DATA_BLOCK "ACESYS_HMI_GROUP"   // DB2
TITLE = ACESYS GROUP DB
{ S7_Optimized_Access := 'FALSE' }
AUTHOR : METIS
FAMILY : ACESYS
NAME : GroupDB
VERSION : 8.0
   VAR
      STATUS : Array[0..500] of "ACESYS_HMI_STAT_32T";   // Group Status to HMI
   END_VAR
BEGIN
   STATUS[0].EXT.AlarmWarnUnAck := FALSE;
   STATUS[0].EXT.AckRequired := FALSE;
   STATUS[0].EXT.Maintanence := FALSE;
   STATUS[0].EXT.Operation := FALSE;
   STATUS[0].EXT.Forced := FALSE;
   STATUS[0].EXT.BIT29 := FALSE;
   STATUS[0].EXT.BIT30 := FALSE;
   STATUS[0].EXT.BIT31 := FALSE;
   STATUS[0].EXT.ModeBit1 := FALSE;
   STATUS[0].EXT.ModeBit2 := FALSE;
   STATUS[0].EXT.ModeBit3 := FALSE;
   STATUS[0].EXT.BIT19 := FALSE;
   STATUS[0].EXT.BIT20 := FALSE;
   STATUS[0].EXT.AlarmSuppressed := FALSE;
   STATUS[0].EXT.AlarmPresent := FALSE;
   STATUS[0].EXT.AlarmFailUnAck := FALSE;
   STATUS[0].Status := 0;
   STATUS[0].TimeStamp := 16#0000;
   STATUS[1].EXT.AlarmWarnUnAck := FALSE;
   STATUS[1].EXT.AckRequired := FALSE;
   STATUS[1].EXT.Maintanence := FALSE;
   STATUS[1].EXT.Operation := FALSE;
   STATUS[1].EXT.Forced := FALSE;
   STATUS[1].EXT.BIT29 := FALSE;
   STATUS[1].EXT.BIT30 := FALSE;
   STATUS[1].EXT.BIT31 := FALSE;
   STATUS[1].EXT.ModeBit1 := FALSE;
   STATUS[1].EXT.ModeBit2 := FALSE;
   STATUS[1].EXT.ModeBit3 := FALSE;
   STATUS[1].EXT.BIT19 := FALSE;
   STATUS[1].EXT.BIT20 := FALSE;
   STATUS[1].EXT.AlarmSuppressed := FALSE;
   STATUS[1].EXT.AlarmPresent := FALSE;
   STATUS[1].EXT.AlarmFailUnAck := FALSE;
   STATUS[1].Status := 8193;
   STATUS[1].TimeStamp := 16#CB75;
   STATUS[2].EXT.AlarmWarnUnAck := FALSE;
   STATUS[2].EXT.AckRequired := FALSE;
   STATUS[2].EXT.Maintanence := FALSE;
   STATUS[2].EXT.Operation := FALSE;
   STATUS[2].EXT.Forced := FALSE;
   STATUS[2].EXT.BIT29 := FALSE;
   STATUS[2].EXT.BIT30 := FALSE;
   STATUS[2].EXT.BIT31 := FALSE;
   STATUS[2].EXT.ModeBit1 := FALSE;
   STATUS[2].EXT.ModeBit2 := FALSE;
   STATUS[2].EXT.ModeBit3 := FALSE;
   STATUS[2].EXT.BIT19 := FALSE;
   STATUS[2].EXT.BIT20 := FALSE;
   STATUS[2].EXT.AlarmSuppressed := FALSE;
   STATUS[2].EXT.AlarmPresent := FALSE;
   STATUS[2].EXT.AlarmFailUnAck := FALSE;
   STATUS[2].Status := 8193;
   STATUS[2].TimeStamp := 16#E395;
   STATUS[3].EXT.AlarmWarnUnAck := FALSE;
   STATUS[3].EXT.AckRequired := FALSE;
   STATUS[3].EXT.Maintanence := FALSE;
   STATUS[3].EXT.Operation := FALSE;
   STATUS[3].EXT.Forced := FALSE;
   STATUS[3].EXT.BIT29 := FALSE;
   STATUS[3].EXT.BIT30 := FALSE;
   STATUS[3].EXT.BIT31 := FALSE;
   STATUS[3].EXT.ModeBit1 := FALSE;
   STATUS[3].EXT.ModeBit2 := FALSE;
   STATUS[3].EXT.ModeBit3 := FALSE;
   STATUS[3].EXT.BIT19 := FALSE;
   STATUS[3].EXT.BIT20 := FALSE;
   STATUS[3].EXT.AlarmSuppressed := FALSE;
   STATUS[3].EXT.AlarmPresent := FALSE;
   STATUS[3].EXT.AlarmFailUnAck := FALSE;
   STATUS[3].Status := 4286;
   STATUS[3].TimeStamp := 16#BB87;
   STATUS[4].EXT.AlarmWarnUnAck := FALSE;
   STATUS[4].EXT.AckRequired := FALSE;
   STATUS[4].EXT.Maintanence := FALSE;
   STATUS[4].EXT.Operation := FALSE;
   STATUS[4].EXT.Forced := FALSE;
   STATUS[4].EXT.BIT29 := FALSE;
   STATUS[4].EXT.BIT30 := FALSE;
   STATUS[4].EXT.BIT31 := FALSE;
   STATUS[4].EXT.ModeBit1 := FALSE;
   STATUS[4].EXT.ModeBit2 := FALSE;
   STATUS[4].EXT.ModeBit3 := FALSE;
   STATUS[4].EXT.BIT19 := FALSE;
   STATUS[4].EXT.BIT20 := FALSE;
   STATUS[4].EXT.AlarmSuppressed := FALSE;
   STATUS[4].EXT.AlarmPresent := FALSE;
   STATUS[4].EXT.AlarmFailUnAck := FALSE;
   STATUS[4].Status := 8215;
   STATUS[4].TimeStamp := 16#CB75;
   STATUS[5].EXT.AlarmWarnUnAck := FALSE;
   STATUS[5].EXT.AckRequired := FALSE;
   STATUS[5].EXT.Maintanence := FALSE;
   STATUS[5].EXT.Operation := FALSE;
   STATUS[5].EXT.Forced := FALSE;
   STATUS[5].EXT.BIT29 := FALSE;
   STATUS[5].EXT.BIT30 := FALSE;
   STATUS[5].EXT.BIT31 := FALSE;
   STATUS[5].EXT.ModeBit1 := FALSE;
   STATUS[5].EXT.ModeBit2 := FALSE;
   STATUS[5].EXT.ModeBit3 := FALSE;
   STATUS[5].EXT.BIT19 := FALSE;
   STATUS[5].EXT.BIT20 := FALSE;
   STATUS[5].EXT.AlarmSuppressed := FALSE;
   STATUS[5].EXT.AlarmPresent := FALSE;
   STATUS[5].EXT.AlarmFailUnAck := FALSE;
   STATUS[5].Status := 8193;
   STATUS[5].TimeStamp := 16#84C0;
   STATUS[6].EXT.AlarmWarnUnAck := FALSE;
   STATUS[6].EXT.AckRequired := FALSE;
   STATUS[6].EXT.Maintanence := FALSE;
   STATUS[6].EXT.Operation := FALSE;
   STATUS[6].EXT.Forced := FALSE;
   STATUS[6].EXT.BIT29 := FALSE;
   STATUS[6].EXT.BIT30 := FALSE;
   STATUS[6].EXT.BIT31 := FALSE;
   STATUS[6].EXT.ModeBit1 := FALSE;
   STATUS[6].EXT.ModeBit2 := FALSE;
   STATUS[6].EXT.ModeBit3 := FALSE;
   STATUS[6].EXT.BIT19 := FALSE;
   STATUS[6].EXT.BIT20 := FALSE;
   STATUS[6].EXT.AlarmSuppressed := FALSE;
   STATUS[6].EXT.AlarmPresent := FALSE;
   STATUS[6].EXT.AlarmFailUnAck := FALSE;
   STATUS[6].Status := 8193;
   STATUS[6].TimeStamp := 16#84BA;
   STATUS[7].EXT.AlarmWarnUnAck := FALSE;
   STATUS[7].EXT.AckRequired := FALSE;
   STATUS[7].EXT.Maintanence := FALSE;
   STATUS[7].EXT.Operation := TRUE;
   STATUS[7].EXT.Forced := FALSE;
   STATUS[7].EXT.BIT29 := FALSE;
   STATUS[7].EXT.BIT30 := FALSE;
   STATUS[7].EXT.BIT31 := FALSE;
   STATUS[7].EXT.ModeBit1 := FALSE;
   STATUS[7].EXT.ModeBit2 := FALSE;
   STATUS[7].EXT.ModeBit3 := FALSE;
   STATUS[7].EXT.BIT19 := FALSE;
   STATUS[7].EXT.BIT20 := FALSE;
   STATUS[7].EXT.AlarmSuppressed := FALSE;
   STATUS[7].EXT.AlarmPresent := FALSE;
   STATUS[7].EXT.AlarmFailUnAck := FALSE;
   STATUS[7].Status := 4104;
   STATUS[7].TimeStamp := 16#C030;
   STATUS[8].EXT.AlarmWarnUnAck := FALSE;
   STATUS[8].EXT.AckRequired := FALSE;
   STATUS[8].EXT.Maintanence := FALSE;
   STATUS[8].EXT.Operation := FALSE;
   STATUS[8].EXT.Forced := FALSE;
   STATUS[8].EXT.BIT29 := FALSE;
   STATUS[8].EXT.BIT30 := FALSE;
   STATUS[8].EXT.BIT31 := FALSE;
   STATUS[8].EXT.ModeBit1 := FALSE;
   STATUS[8].EXT.ModeBit2 := FALSE;
   STATUS[8].EXT.ModeBit3 := FALSE;
   STATUS[8].EXT.BIT19 := FALSE;
   STATUS[8].EXT.BIT20 := FALSE;
   STATUS[8].EXT.AlarmSuppressed := FALSE;
   STATUS[8].EXT.AlarmPresent := FALSE;
   STATUS[8].EXT.AlarmFailUnAck := FALSE;
   STATUS[8].Status := 8193;
   STATUS[8].TimeStamp := 16#60BB;
   STATUS[9].EXT.AlarmWarnUnAck := FALSE;
   STATUS[9].EXT.AckRequired := FALSE;
   STATUS[9].EXT.Maintanence := FALSE;
   STATUS[9].EXT.Operation := FALSE;
   STATUS[9].EXT.Forced := FALSE;
   STATUS[9].EXT.BIT29 := FALSE;
   STATUS[9].EXT.BIT30 := FALSE;
   STATUS[9].EXT.BIT31 := FALSE;
   STATUS[9].EXT.ModeBit1 := FALSE;
   STATUS[9].EXT.ModeBit2 := FALSE;
   STATUS[9].EXT.ModeBit3 := FALSE;
   STATUS[9].EXT.BIT19 := FALSE;
   STATUS[9].EXT.BIT20 := FALSE;
   STATUS[9].EXT.AlarmSuppressed := FALSE;
   STATUS[9].EXT.AlarmPresent := FALSE;
   STATUS[9].EXT.AlarmFailUnAck := FALSE;
   STATUS[9].Status := 8193;
   STATUS[9].TimeStamp := 16#60BB;
   STATUS[10].EXT.AlarmWarnUnAck := FALSE;
   STATUS[10].EXT.AckRequired := FALSE;
   STATUS[10].EXT.Maintanence := FALSE;
   STATUS[10].EXT.Operation := FALSE;
   STATUS[10].EXT.Forced := FALSE;
   STATUS[10].EXT.BIT29 := FALSE;
   STATUS[10].EXT.BIT30 := FALSE;
   STATUS[10].EXT.BIT31 := FALSE;
   STATUS[10].EXT.ModeBit1 := FALSE;
   STATUS[10].EXT.ModeBit2 := FALSE;
   STATUS[10].EXT.ModeBit3 := FALSE;
   STATUS[10].EXT.BIT19 := FALSE;
   STATUS[10].EXT.BIT20 := FALSE;
   STATUS[10].EXT.AlarmSuppressed := FALSE;
   STATUS[10].EXT.AlarmPresent := FALSE;
   STATUS[10].EXT.AlarmFailUnAck := FALSE;
   STATUS[10].Status := 8193;
   STATUS[10].TimeStamp := 16#60BB;
   STATUS[11].EXT.AlarmWarnUnAck := FALSE;
   STATUS[11].EXT.AckRequired := FALSE;
   STATUS[11].EXT.Maintanence := FALSE;
   STATUS[11].EXT.Operation := FALSE;
   STATUS[11].EXT.Forced := FALSE;
   STATUS[11].EXT.BIT29 := FALSE;
   STATUS[11].EXT.BIT30 := FALSE;
   STATUS[11].EXT.BIT31 := FALSE;
   STATUS[11].EXT.ModeBit1 := FALSE;
   STATUS[11].EXT.ModeBit2 := FALSE;
   STATUS[11].EXT.ModeBit3 := FALSE;
   STATUS[11].EXT.BIT19 := FALSE;
   STATUS[11].EXT.BIT20 := FALSE;
   STATUS[11].EXT.AlarmSuppressed := FALSE;
   STATUS[11].EXT.AlarmPresent := FALSE;
   STATUS[11].EXT.AlarmFailUnAck := FALSE;
   STATUS[11].Status := 8193;
   STATUS[11].TimeStamp := 16#60BB;
   STATUS[12].EXT.AlarmWarnUnAck := FALSE;
   STATUS[12].EXT.AckRequired := FALSE;
   STATUS[12].EXT.Maintanence := FALSE;
   STATUS[12].EXT.Operation := FALSE;
   STATUS[12].EXT.Forced := FALSE;
   STATUS[12].EXT.BIT29 := FALSE;
   STATUS[12].EXT.BIT30 := FALSE;
   STATUS[12].EXT.BIT31 := FALSE;
   STATUS[12].EXT.ModeBit1 := FALSE;
   STATUS[12].EXT.ModeBit2 := FALSE;
   STATUS[12].EXT.ModeBit3 := FALSE;
   STATUS[12].EXT.BIT19 := FALSE;
   STATUS[12].EXT.BIT20 := FALSE;
   STATUS[12].EXT.AlarmSuppressed := FALSE;
   STATUS[12].EXT.AlarmPresent := FALSE;
   STATUS[12].EXT.AlarmFailUnAck := FALSE;
   STATUS[12].Status := 8193;
   STATUS[12].TimeStamp := 16#60BB;
   STATUS[13].EXT.AlarmWarnUnAck := FALSE;
   STATUS[13].EXT.AckRequired := FALSE;
   STATUS[13].EXT.Maintanence := FALSE;
   STATUS[13].EXT.Operation := FALSE;
   STATUS[13].EXT.Forced := FALSE;
   STATUS[13].EXT.BIT29 := FALSE;
   STATUS[13].EXT.BIT30 := FALSE;
   STATUS[13].EXT.BIT31 := FALSE;
   STATUS[13].EXT.ModeBit1 := FALSE;
   STATUS[13].EXT.ModeBit2 := FALSE;
   STATUS[13].EXT.ModeBit3 := FALSE;
   STATUS[13].EXT.BIT19 := FALSE;
   STATUS[13].EXT.BIT20 := FALSE;
   STATUS[13].EXT.AlarmSuppressed := FALSE;
   STATUS[13].EXT.AlarmPresent := FALSE;
   STATUS[13].EXT.AlarmFailUnAck := FALSE;
   STATUS[13].Status := 8193;
   STATUS[13].TimeStamp := 16#60BB;
   STATUS[14].EXT.AlarmWarnUnAck := FALSE;
   STATUS[14].EXT.AckRequired := FALSE;
   STATUS[14].EXT.Maintanence := FALSE;
   STATUS[14].EXT.Operation := FALSE;
   STATUS[14].EXT.Forced := FALSE;
   STATUS[14].EXT.BIT29 := FALSE;
   STATUS[14].EXT.BIT30 := FALSE;
   STATUS[14].EXT.BIT31 := FALSE;
   STATUS[14].EXT.ModeBit1 := FALSE;
   STATUS[14].EXT.ModeBit2 := FALSE;
   STATUS[14].EXT.ModeBit3 := FALSE;
   STATUS[14].EXT.BIT19 := FALSE;
   STATUS[14].EXT.BIT20 := FALSE;
   STATUS[14].EXT.AlarmSuppressed := FALSE;
   STATUS[14].EXT.AlarmPresent := FALSE;
   STATUS[14].EXT.AlarmFailUnAck := FALSE;
   STATUS[14].Status := 8193;
   STATUS[14].TimeStamp := 16#60BB;
   STATUS[15].EXT.AlarmWarnUnAck := FALSE;
   STATUS[15].EXT.AckRequired := FALSE;
   STATUS[15].EXT.Maintanence := FALSE;
   STATUS[15].EXT.Operation := FALSE;
   STATUS[15].EXT.Forced := FALSE;
   STATUS[15].EXT.BIT29 := FALSE;
   STATUS[15].EXT.BIT30 := FALSE;
   STATUS[15].EXT.BIT31 := FALSE;
   STATUS[15].EXT.ModeBit1 := FALSE;
   STATUS[15].EXT.ModeBit2 := FALSE;
   STATUS[15].EXT.ModeBit3 := FALSE;
   STATUS[15].EXT.BIT19 := FALSE;
   STATUS[15].EXT.BIT20 := FALSE;
   STATUS[15].EXT.AlarmSuppressed := FALSE;
   STATUS[15].EXT.AlarmPresent := FALSE;
   STATUS[15].EXT.AlarmFailUnAck := FALSE;
   STATUS[15].Status := 8193;
   STATUS[15].TimeStamp := 16#60BB;
   STATUS[16].EXT.AlarmWarnUnAck := FALSE;
   STATUS[16].EXT.AckRequired := FALSE;
   STATUS[16].EXT.Maintanence := FALSE;
   STATUS[16].EXT.Operation := FALSE;
   STATUS[16].EXT.Forced := FALSE;
   STATUS[16].EXT.BIT29 := FALSE;
   STATUS[16].EXT.BIT30 := FALSE;
   STATUS[16].EXT.BIT31 := FALSE;
   STATUS[16].EXT.ModeBit1 := FALSE;
   STATUS[16].EXT.ModeBit2 := FALSE;
   STATUS[16].EXT.ModeBit3 := FALSE;
   STATUS[16].EXT.BIT19 := FALSE;
   STATUS[16].EXT.BIT20 := FALSE;
   STATUS[16].EXT.AlarmSuppressed := FALSE;
   STATUS[16].EXT.AlarmPresent := FALSE;
   STATUS[16].EXT.AlarmFailUnAck := FALSE;
   STATUS[16].Status := 0;
   STATUS[16].TimeStamp := 16#0000;
   STATUS[17].EXT.AlarmWarnUnAck := FALSE;
   STATUS[17].EXT.AckRequired := FALSE;
   STATUS[17].EXT.Maintanence := FALSE;
   STATUS[17].EXT.Operation := FALSE;
   STATUS[17].EXT.Forced := FALSE;
   STATUS[17].EXT.BIT29 := FALSE;
   STATUS[17].EXT.BIT30 := FALSE;
   STATUS[17].EXT.BIT31 := FALSE;
   STATUS[17].EXT.ModeBit1 := FALSE;
   STATUS[17].EXT.ModeBit2 := FALSE;
   STATUS[17].EXT.ModeBit3 := FALSE;
   STATUS[17].EXT.BIT19 := FALSE;
   STATUS[17].EXT.BIT20 := FALSE;
   STATUS[17].EXT.AlarmSuppressed := FALSE;
   STATUS[17].EXT.AlarmPresent := FALSE;
   STATUS[17].EXT.AlarmFailUnAck := FALSE;
   STATUS[17].Status := 0;
   STATUS[17].TimeStamp := 16#0000;
   STATUS[18].EXT.AlarmWarnUnAck := FALSE;
   STATUS[18].EXT.AckRequired := FALSE;
   STATUS[18].EXT.Maintanence := FALSE;
   STATUS[18].EXT.Operation := FALSE;
   STATUS[18].EXT.Forced := FALSE;
   STATUS[18].EXT.BIT29 := FALSE;
   STATUS[18].EXT.BIT30 := FALSE;
   STATUS[18].EXT.BIT31 := FALSE;
   STATUS[18].EXT.ModeBit1 := FALSE;
   STATUS[18].EXT.ModeBit2 := FALSE;
   STATUS[18].EXT.ModeBit3 := FALSE;
   STATUS[18].EXT.BIT19 := FALSE;
   STATUS[18].EXT.BIT20 := FALSE;
   STATUS[18].EXT.AlarmSuppressed := FALSE;
   STATUS[18].EXT.AlarmPresent := FALSE;
   STATUS[18].EXT.AlarmFailUnAck := FALSE;
   STATUS[18].Status := 0;
   STATUS[18].TimeStamp := 16#0000;
   STATUS[19].EXT.AlarmWarnUnAck := FALSE;
   STATUS[19].EXT.AckRequired := FALSE;
   STATUS[19].EXT.Maintanence := FALSE;
   STATUS[19].EXT.Operation := FALSE;
   STATUS[19].EXT.Forced := FALSE;
   STATUS[19].EXT.BIT29 := FALSE;
   STATUS[19].EXT.BIT30 := FALSE;
   STATUS[19].EXT.BIT31 := FALSE;
   STATUS[19].EXT.ModeBit1 := FALSE;
   STATUS[19].EXT.ModeBit2 := FALSE;
   STATUS[19].EXT.ModeBit3 := FALSE;
   STATUS[19].EXT.BIT19 := FALSE;
   STATUS[19].EXT.BIT20 := FALSE;
   STATUS[19].EXT.AlarmSuppressed := FALSE;
   STATUS[19].EXT.AlarmPresent := FALSE;
   STATUS[19].EXT.AlarmFailUnAck := FALSE;
   STATUS[19].Status := 0;
   STATUS[19].TimeStamp := 16#0000;
   STATUS[20].EXT.AlarmWarnUnAck := FALSE;
   STATUS[20].EXT.AckRequired := FALSE;
   STATUS[20].EXT.Maintanence := FALSE;
   STATUS[20].EXT.Operation := FALSE;
   STATUS[20].EXT.Forced := FALSE;
   STATUS[20].EXT.BIT29 := FALSE;
   STATUS[20].EXT.BIT30 := FALSE;
   STATUS[20].EXT.BIT31 := FALSE;
   STATUS[20].EXT.ModeBit1 := FALSE;
   STATUS[20].EXT.ModeBit2 := FALSE;
   STATUS[20].EXT.ModeBit3 := FALSE;
   STATUS[20].EXT.BIT19 := FALSE;
   STATUS[20].EXT.BIT20 := FALSE;
   STATUS[20].EXT.AlarmSuppressed := FALSE;
   STATUS[20].EXT.AlarmPresent := FALSE;
   STATUS[20].EXT.AlarmFailUnAck := FALSE;
   STATUS[20].Status := 0;
   STATUS[20].TimeStamp := 16#0000;
   STATUS[21].EXT.AlarmWarnUnAck := FALSE;
   STATUS[21].EXT.AckRequired := FALSE;
   STATUS[21].EXT.Maintanence := FALSE;
   STATUS[21].EXT.Operation := FALSE;
   STATUS[21].EXT.Forced := FALSE;
   STATUS[21].EXT.BIT29 := FALSE;
   STATUS[21].EXT.BIT30 := FALSE;
   STATUS[21].EXT.BIT31 := FALSE;
   STATUS[21].EXT.ModeBit1 := FALSE;
   STATUS[21].EXT.ModeBit2 := FALSE;
   STATUS[21].EXT.ModeBit3 := FALSE;
   STATUS[21].EXT.BIT19 := FALSE;
   STATUS[21].EXT.BIT20 := FALSE;
   STATUS[21].EXT.AlarmSuppressed := FALSE;
   STATUS[21].EXT.AlarmPresent := FALSE;
   STATUS[21].EXT.AlarmFailUnAck := FALSE;
   STATUS[21].Status := 0;
   STATUS[21].TimeStamp := 16#0000;
   STATUS[22].EXT.AlarmWarnUnAck := FALSE;
   STATUS[22].EXT.AckRequired := FALSE;
   STATUS[22].EXT.Maintanence := FALSE;
   STATUS[22].EXT.Operation := FALSE;
   STATUS[22].EXT.Forced := FALSE;
   STATUS[22].EXT.BIT29 := FALSE;
   STATUS[22].EXT.BIT30 := FALSE;
   STATUS[22].EXT.BIT31 := FALSE;
   STATUS[22].EXT.ModeBit1 := FALSE;
   STATUS[22].EXT.ModeBit2 := FALSE;
   STATUS[22].EXT.ModeBit3 := FALSE;
   STATUS[22].EXT.BIT19 := FALSE;
   STATUS[22].EXT.BIT20 := FALSE;
   STATUS[22].EXT.AlarmSuppressed := FALSE;
   STATUS[22].EXT.AlarmPresent := FALSE;
   STATUS[22].EXT.AlarmFailUnAck := FALSE;
   STATUS[22].Status := 0;
   STATUS[22].TimeStamp := 16#0000;
   STATUS[23].EXT.AlarmWarnUnAck := FALSE;
   STATUS[23].EXT.AckRequired := FALSE;
   STATUS[23].EXT.Maintanence := FALSE;
   STATUS[23].EXT.Operation := FALSE;
   STATUS[23].EXT.Forced := FALSE;
   STATUS[23].EXT.BIT29 := FALSE;
   STATUS[23].EXT.BIT30 := FALSE;
   STATUS[23].EXT.BIT31 := FALSE;
   STATUS[23].EXT.ModeBit1 := FALSE;
   STATUS[23].EXT.ModeBit2 := FALSE;
   STATUS[23].EXT.ModeBit3 := FALSE;
   STATUS[23].EXT.BIT19 := FALSE;
   STATUS[23].EXT.BIT20 := FALSE;
   STATUS[23].EXT.AlarmSuppressed := FALSE;
   STATUS[23].EXT.AlarmPresent := FALSE;
   STATUS[23].EXT.AlarmFailUnAck := FALSE;
   STATUS[23].Status := 0;
   STATUS[23].TimeStamp := 16#0000;
   STATUS[24].EXT.AlarmWarnUnAck := FALSE;
   STATUS[24].EXT.AckRequired := FALSE;
   STATUS[24].EXT.Maintanence := FALSE;
   STATUS[24].EXT.Operation := FALSE;
   STATUS[24].EXT.Forced := FALSE;
   STATUS[24].EXT.BIT29 := FALSE;
   STATUS[24].EXT.BIT30 := FALSE;
   STATUS[24].EXT.BIT31 := FALSE;
   STATUS[24].EXT.ModeBit1 := FALSE;
   STATUS[24].EXT.ModeBit2 := FALSE;
   STATUS[24].EXT.ModeBit3 := FALSE;
   STATUS[24].EXT.BIT19 := FALSE;
   STATUS[24].EXT.BIT20 := FALSE;
   STATUS[24].EXT.AlarmSuppressed := FALSE;
   STATUS[24].EXT.AlarmPresent := FALSE;
   STATUS[24].EXT.AlarmFailUnAck := FALSE;
   STATUS[24].Status := 0;
   STATUS[24].TimeStamp := 16#0000;
   STATUS[25].EXT.AlarmWarnUnAck := FALSE;
   STATUS[25].EXT.AckRequired := FALSE;
   STATUS[25].EXT.Maintanence := FALSE;
   STATUS[25].EXT.Operation := FALSE;
   STATUS[25].EXT.Forced := FALSE;
   STATUS[25].EXT.BIT29 := FALSE;
   STATUS[25].EXT.BIT30 := FALSE;
   STATUS[25].EXT.BIT31 := FALSE;
   STATUS[25].EXT.ModeBit1 := FALSE;
   STATUS[25].EXT.ModeBit2 := FALSE;
   STATUS[25].EXT.ModeBit3 := FALSE;
   STATUS[25].EXT.BIT19 := FALSE;
   STATUS[25].EXT.BIT20 := FALSE;
   STATUS[25].EXT.AlarmSuppressed := FALSE;
   STATUS[25].EXT.AlarmPresent := FALSE;
   STATUS[25].EXT.AlarmFailUnAck := FALSE;
   STATUS[25].Status := 0;
   STATUS[25].TimeStamp := 16#0000;
   STATUS[26].EXT.AlarmWarnUnAck := FALSE;
   STATUS[26].EXT.AckRequired := FALSE;
   STATUS[26].EXT.Maintanence := FALSE;
   STATUS[26].EXT.Operation := FALSE;
   STATUS[26].EXT.Forced := FALSE;
   STATUS[26].EXT.BIT29 := FALSE;
   STATUS[26].EXT.BIT30 := FALSE;
   STATUS[26].EXT.BIT31 := FALSE;
   STATUS[26].EXT.ModeBit1 := FALSE;
   STATUS[26].EXT.ModeBit2 := FALSE;
   STATUS[26].EXT.ModeBit3 := FALSE;
   STATUS[26].EXT.BIT19 := FALSE;
   STATUS[26].EXT.BIT20 := FALSE;
   STATUS[26].EXT.AlarmSuppressed := FALSE;
   STATUS[26].EXT.AlarmPresent := FALSE;
   STATUS[26].EXT.AlarmFailUnAck := FALSE;
   STATUS[26].Status := 0;
   STATUS[26].TimeStamp := 16#0000;
   STATUS[27].EXT.AlarmWarnUnAck := FALSE;
   STATUS[27].EXT.AckRequired := FALSE;
   STATUS[27].EXT.Maintanence := FALSE;
   STATUS[27].EXT.Operation := FALSE;
   STATUS[27].EXT.Forced := FALSE;
   STATUS[27].EXT.BIT29 := FALSE;
   STATUS[27].EXT.BIT30 := FALSE;
   STATUS[27].EXT.BIT31 := FALSE;
   STATUS[27].EXT.ModeBit1 := FALSE;
   STATUS[27].EXT.ModeBit2 := FALSE;
   STATUS[27].EXT.ModeBit3 := FALSE;
   STATUS[27].EXT.BIT19 := FALSE;
   STATUS[27].EXT.BIT20 := FALSE;
   STATUS[27].EXT.AlarmSuppressed := FALSE;
   STATUS[27].EXT.AlarmPresent := FALSE;
   STATUS[27].EXT.AlarmFailUnAck := FALSE;
   STATUS[27].Status := 0;
   STATUS[27].TimeStamp := 16#0000;
   STATUS[28].EXT.AlarmWarnUnAck := FALSE;
   STATUS[28].EXT.AckRequired := FALSE;
   STATUS[28].EXT.Maintanence := FALSE;
   STATUS[28].EXT.Operation := FALSE;
   STATUS[28].EXT.Forced := FALSE;
   STATUS[28].EXT.BIT29 := FALSE;
   STATUS[28].EXT.BIT30 := FALSE;
   STATUS[28].EXT.BIT31 := FALSE;
   STATUS[28].EXT.ModeBit1 := FALSE;
   STATUS[28].EXT.ModeBit2 := FALSE;
   STATUS[28].EXT.ModeBit3 := FALSE;
   STATUS[28].EXT.BIT19 := FALSE;
   STATUS[28].EXT.BIT20 := FALSE;
   STATUS[28].EXT.AlarmSuppressed := FALSE;
   STATUS[28].EXT.AlarmPresent := FALSE;
   STATUS[28].EXT.AlarmFailUnAck := FALSE;
   STATUS[28].Status := 0;
   STATUS[28].TimeStamp := 16#0000;
   STATUS[29].EXT.AlarmWarnUnAck := FALSE;
   STATUS[29].EXT.AckRequired := FALSE;
   STATUS[29].EXT.Maintanence := FALSE;
   STATUS[29].EXT.Operation := FALSE;
   STATUS[29].EXT.Forced := FALSE;
   STATUS[29].EXT.BIT29 := FALSE;
   STATUS[29].EXT.BIT30 := FALSE;
   STATUS[29].EXT.BIT31 := FALSE;
   STATUS[29].EXT.ModeBit1 := FALSE;
   STATUS[29].EXT.ModeBit2 := FALSE;
   STATUS[29].EXT.ModeBit3 := FALSE;
   STATUS[29].EXT.BIT19 := FALSE;
   STATUS[29].EXT.BIT20 := FALSE;
   STATUS[29].EXT.AlarmSuppressed := FALSE;
   STATUS[29].EXT.AlarmPresent := FALSE;
   STATUS[29].EXT.AlarmFailUnAck := FALSE;
   STATUS[29].Status := 0;
   STATUS[29].TimeStamp := 16#0000;
   STATUS[30].EXT.AlarmWarnUnAck := FALSE;
   STATUS[30].EXT.AckRequired := FALSE;
   STATUS[30].EXT.Maintanence := FALSE;
   STATUS[30].EXT.Operation := FALSE;
   STATUS[30].EXT.Forced := FALSE;
   STATUS[30].EXT.BIT29 := FALSE;
   STATUS[30].EXT.BIT30 := FALSE;
   STATUS[30].EXT.BIT31 := FALSE;
   STATUS[30].EXT.ModeBit1 := FALSE;
   STATUS[30].EXT.ModeBit2 := FALSE;
   STATUS[30].EXT.ModeBit3 := FALSE;
   STATUS[30].EXT.BIT19 := FALSE;
   STATUS[30].EXT.BIT20 := FALSE;
   STATUS[30].EXT.AlarmSuppressed := FALSE;
   STATUS[30].EXT.AlarmPresent := FALSE;
   STATUS[30].EXT.AlarmFailUnAck := FALSE;
   STATUS[30].Status := 0;
   STATUS[30].TimeStamp := 16#0000;
   STATUS[31].EXT.AlarmWarnUnAck := FALSE;
   STATUS[31].EXT.AckRequired := FALSE;
   STATUS[31].EXT.Maintanence := FALSE;
   STATUS[31].EXT.Operation := FALSE;
   STATUS[31].EXT.Forced := FALSE;
   STATUS[31].EXT.BIT29 := FALSE;
   STATUS[31].EXT.BIT30 := FALSE;
   STATUS[31].EXT.BIT31 := FALSE;
   STATUS[31].EXT.ModeBit1 := FALSE;
   STATUS[31].EXT.ModeBit2 := FALSE;
   STATUS[31].EXT.ModeBit3 := FALSE;
   STATUS[31].EXT.BIT19 := FALSE;
   STATUS[31].EXT.BIT20 := FALSE;
   STATUS[31].EXT.AlarmSuppressed := FALSE;
   STATUS[31].EXT.AlarmPresent := FALSE;
   STATUS[31].EXT.AlarmFailUnAck := FALSE;
   STATUS[31].Status := 0;
   STATUS[31].TimeStamp := 16#0000;
   STATUS[32].EXT.AlarmWarnUnAck := FALSE;
   STATUS[32].EXT.AckRequired := FALSE;
   STATUS[32].EXT.Maintanence := FALSE;
   STATUS[32].EXT.Operation := FALSE;
   STATUS[32].EXT.Forced := FALSE;
   STATUS[32].EXT.BIT29 := FALSE;
   STATUS[32].EXT.BIT30 := FALSE;
   STATUS[32].EXT.BIT31 := FALSE;
   STATUS[32].EXT.ModeBit1 := FALSE;
   STATUS[32].EXT.ModeBit2 := FALSE;
   STATUS[32].EXT.ModeBit3 := FALSE;
   STATUS[32].EXT.BIT19 := FALSE;
   STATUS[32].EXT.BIT20 := FALSE;
   STATUS[32].EXT.AlarmSuppressed := FALSE;
   STATUS[32].EXT.AlarmPresent := FALSE;
   STATUS[32].EXT.AlarmFailUnAck := FALSE;
   STATUS[32].Status := 0;
   STATUS[32].TimeStamp := 16#0000;
   STATUS[33].EXT.AlarmWarnUnAck := FALSE;
   STATUS[33].EXT.AckRequired := FALSE;
   STATUS[33].EXT.Maintanence := FALSE;
   STATUS[33].EXT.Operation := FALSE;
   STATUS[33].EXT.Forced := FALSE;
   STATUS[33].EXT.BIT29 := FALSE;
   STATUS[33].EXT.BIT30 := FALSE;
   STATUS[33].EXT.BIT31 := FALSE;
   STATUS[33].EXT.ModeBit1 := FALSE;
   STATUS[33].EXT.ModeBit2 := FALSE;
   STATUS[33].EXT.ModeBit3 := FALSE;
   STATUS[33].EXT.BIT19 := FALSE;
   STATUS[33].EXT.BIT20 := FALSE;
   STATUS[33].EXT.AlarmSuppressed := FALSE;
   STATUS[33].EXT.AlarmPresent := FALSE;
   STATUS[33].EXT.AlarmFailUnAck := FALSE;
   STATUS[33].Status := 0;
   STATUS[33].TimeStamp := 16#0000;
   STATUS[34].EXT.AlarmWarnUnAck := FALSE;
   STATUS[34].EXT.AckRequired := FALSE;
   STATUS[34].EXT.Maintanence := FALSE;
   STATUS[34].EXT.Operation := FALSE;
   STATUS[34].EXT.Forced := FALSE;
   STATUS[34].EXT.BIT29 := FALSE;
   STATUS[34].EXT.BIT30 := FALSE;
   STATUS[34].EXT.BIT31 := FALSE;
   STATUS[34].EXT.ModeBit1 := FALSE;
   STATUS[34].EXT.ModeBit2 := FALSE;
   STATUS[34].EXT.ModeBit3 := FALSE;
   STATUS[34].EXT.BIT19 := FALSE;
   STATUS[34].EXT.BIT20 := FALSE;
   STATUS[34].EXT.AlarmSuppressed := FALSE;
   STATUS[34].EXT.AlarmPresent := FALSE;
   STATUS[34].EXT.AlarmFailUnAck := FALSE;
   STATUS[34].Status := 0;
   STATUS[34].TimeStamp := 16#0000;
   STATUS[35].EXT.AlarmWarnUnAck := FALSE;
   STATUS[35].EXT.AckRequired := FALSE;
   STATUS[35].EXT.Maintanence := FALSE;
   STATUS[35].EXT.Operation := FALSE;
   STATUS[35].EXT.Forced := FALSE;
   STATUS[35].EXT.BIT29 := FALSE;
   STATUS[35].EXT.BIT30 := FALSE;
   STATUS[35].EXT.BIT31 := FALSE;
   STATUS[35].EXT.ModeBit1 := FALSE;
   STATUS[35].EXT.ModeBit2 := FALSE;
   STATUS[35].EXT.ModeBit3 := FALSE;
   STATUS[35].EXT.BIT19 := FALSE;
   STATUS[35].EXT.BIT20 := FALSE;
   STATUS[35].EXT.AlarmSuppressed := FALSE;
   STATUS[35].EXT.AlarmPresent := FALSE;
   STATUS[35].EXT.AlarmFailUnAck := FALSE;
   STATUS[35].Status := 0;
   STATUS[35].TimeStamp := 16#0000;
   STATUS[36].EXT.AlarmWarnUnAck := FALSE;
   STATUS[36].EXT.AckRequired := FALSE;
   STATUS[36].EXT.Maintanence := FALSE;
   STATUS[36].EXT.Operation := FALSE;
   STATUS[36].EXT.Forced := FALSE;
   STATUS[36].EXT.BIT29 := FALSE;
   STATUS[36].EXT.BIT30 := FALSE;
   STATUS[36].EXT.BIT31 := FALSE;
   STATUS[36].EXT.ModeBit1 := FALSE;
   STATUS[36].EXT.ModeBit2 := FALSE;
   STATUS[36].EXT.ModeBit3 := FALSE;
   STATUS[36].EXT.BIT19 := FALSE;
   STATUS[36].EXT.BIT20 := FALSE;
   STATUS[36].EXT.AlarmSuppressed := FALSE;
   STATUS[36].EXT.AlarmPresent := FALSE;
   STATUS[36].EXT.AlarmFailUnAck := FALSE;
   STATUS[36].Status := 0;
   STATUS[36].TimeStamp := 16#0000;
   STATUS[37].EXT.AlarmWarnUnAck := FALSE;
   STATUS[37].EXT.AckRequired := FALSE;
   STATUS[37].EXT.Maintanence := FALSE;
   STATUS[37].EXT.Operation := FALSE;
   STATUS[37].EXT.Forced := FALSE;
   STATUS[37].EXT.BIT29 := FALSE;
   STATUS[37].EXT.BIT30 := FALSE;
   STATUS[37].EXT.BIT31 := FALSE;
   STATUS[37].EXT.ModeBit1 := FALSE;
   STATUS[37].EXT.ModeBit2 := FALSE;
   STATUS[37].EXT.ModeBit3 := FALSE;
   STATUS[37].EXT.BIT19 := FALSE;
   STATUS[37].EXT.BIT20 := FALSE;
   STATUS[37].EXT.AlarmSuppressed := FALSE;
   STATUS[37].EXT.AlarmPresent := FALSE;
   STATUS[37].EXT.AlarmFailUnAck := FALSE;
   STATUS[37].Status := 0;
   STATUS[37].TimeStamp := 16#0000;
   STATUS[38].EXT.AlarmWarnUnAck := FALSE;
   STATUS[38].EXT.AckRequired := FALSE;
   STATUS[38].EXT.Maintanence := FALSE;
   STATUS[38].EXT.Operation := FALSE;
   STATUS[38].EXT.Forced := FALSE;
   STATUS[38].EXT.BIT29 := FALSE;
   STATUS[38].EXT.BIT30 := FALSE;
   STATUS[38].EXT.BIT31 := FALSE;
   STATUS[38].EXT.ModeBit1 := FALSE;
   STATUS[38].EXT.ModeBit2 := FALSE;
   STATUS[38].EXT.ModeBit3 := FALSE;
   STATUS[38].EXT.BIT19 := FALSE;
   STATUS[38].EXT.BIT20 := FALSE;
   STATUS[38].EXT.AlarmSuppressed := FALSE;
   STATUS[38].EXT.AlarmPresent := FALSE;
   STATUS[38].EXT.AlarmFailUnAck := FALSE;
   STATUS[38].Status := 0;
   STATUS[38].TimeStamp := 16#0000;
   STATUS[39].EXT.AlarmWarnUnAck := FALSE;
   STATUS[39].EXT.AckRequired := FALSE;
   STATUS[39].EXT.Maintanence := FALSE;
   STATUS[39].EXT.Operation := FALSE;
   STATUS[39].EXT.Forced := FALSE;
   STATUS[39].EXT.BIT29 := FALSE;
   STATUS[39].EXT.BIT30 := FALSE;
   STATUS[39].EXT.BIT31 := FALSE;
   STATUS[39].EXT.ModeBit1 := FALSE;
   STATUS[39].EXT.ModeBit2 := FALSE;
   STATUS[39].EXT.ModeBit3 := FALSE;
   STATUS[39].EXT.BIT19 := FALSE;
   STATUS[39].EXT.BIT20 := FALSE;
   STATUS[39].EXT.AlarmSuppressed := FALSE;
   STATUS[39].EXT.AlarmPresent := FALSE;
   STATUS[39].EXT.AlarmFailUnAck := FALSE;
   STATUS[39].Status := 0;
   STATUS[39].TimeStamp := 16#0000;
   STATUS[40].EXT.AlarmWarnUnAck := FALSE;
   STATUS[40].EXT.AckRequired := FALSE;
   STATUS[40].EXT.Maintanence := FALSE;
   STATUS[40].EXT.Operation := FALSE;
   STATUS[40].EXT.Forced := FALSE;
   STATUS[40].EXT.BIT29 := FALSE;
   STATUS[40].EXT.BIT30 := FALSE;
   STATUS[40].EXT.BIT31 := FALSE;
   STATUS[40].EXT.ModeBit1 := FALSE;
   STATUS[40].EXT.ModeBit2 := FALSE;
   STATUS[40].EXT.ModeBit3 := FALSE;
   STATUS[40].EXT.BIT19 := FALSE;
   STATUS[40].EXT.BIT20 := FALSE;
   STATUS[40].EXT.AlarmSuppressed := FALSE;
   STATUS[40].EXT.AlarmPresent := FALSE;
   STATUS[40].EXT.AlarmFailUnAck := FALSE;
   STATUS[40].Status := 0;
   STATUS[40].TimeStamp := 16#0000;
   STATUS[41].EXT.AlarmWarnUnAck := FALSE;
   STATUS[41].EXT.AckRequired := FALSE;
   STATUS[41].EXT.Maintanence := FALSE;
   STATUS[41].EXT.Operation := FALSE;
   STATUS[41].EXT.Forced := FALSE;
   STATUS[41].EXT.BIT29 := FALSE;
   STATUS[41].EXT.BIT30 := FALSE;
   STATUS[41].EXT.BIT31 := FALSE;
   STATUS[41].EXT.ModeBit1 := FALSE;
   STATUS[41].EXT.ModeBit2 := FALSE;
   STATUS[41].EXT.ModeBit3 := FALSE;
   STATUS[41].EXT.BIT19 := FALSE;
   STATUS[41].EXT.BIT20 := FALSE;
   STATUS[41].EXT.AlarmSuppressed := FALSE;
   STATUS[41].EXT.AlarmPresent := FALSE;
   STATUS[41].EXT.AlarmFailUnAck := FALSE;
   STATUS[41].Status := 0;
   STATUS[41].TimeStamp := 16#0000;
   STATUS[42].EXT.AlarmWarnUnAck := FALSE;
   STATUS[42].EXT.AckRequired := FALSE;
   STATUS[42].EXT.Maintanence := FALSE;
   STATUS[42].EXT.Operation := FALSE;
   STATUS[42].EXT.Forced := FALSE;
   STATUS[42].EXT.BIT29 := FALSE;
   STATUS[42].EXT.BIT30 := FALSE;
   STATUS[42].EXT.BIT31 := FALSE;
   STATUS[42].EXT.ModeBit1 := FALSE;
   STATUS[42].EXT.ModeBit2 := FALSE;
   STATUS[42].EXT.ModeBit3 := FALSE;
   STATUS[42].EXT.BIT19 := FALSE;
   STATUS[42].EXT.BIT20 := FALSE;
   STATUS[42].EXT.AlarmSuppressed := FALSE;
   STATUS[42].EXT.AlarmPresent := FALSE;
   STATUS[42].EXT.AlarmFailUnAck := FALSE;
   STATUS[42].Status := 0;
   STATUS[42].TimeStamp := 16#0000;
   STATUS[43].EXT.AlarmWarnUnAck := FALSE;
   STATUS[43].EXT.AckRequired := FALSE;
   STATUS[43].EXT.Maintanence := FALSE;
   STATUS[43].EXT.Operation := FALSE;
   STATUS[43].EXT.Forced := FALSE;
   STATUS[43].EXT.BIT29 := FALSE;
   STATUS[43].EXT.BIT30 := FALSE;
   STATUS[43].EXT.BIT31 := FALSE;
   STATUS[43].EXT.ModeBit1 := FALSE;
   STATUS[43].EXT.ModeBit2 := FALSE;
   STATUS[43].EXT.ModeBit3 := FALSE;
   STATUS[43].EXT.BIT19 := FALSE;
   STATUS[43].EXT.BIT20 := FALSE;
   STATUS[43].EXT.AlarmSuppressed := FALSE;
   STATUS[43].EXT.AlarmPresent := FALSE;
   STATUS[43].EXT.AlarmFailUnAck := FALSE;
   STATUS[43].Status := 0;
   STATUS[43].TimeStamp := 16#0000;
   STATUS[44].EXT.AlarmWarnUnAck := FALSE;
   STATUS[44].EXT.AckRequired := FALSE;
   STATUS[44].EXT.Maintanence := FALSE;
   STATUS[44].EXT.Operation := FALSE;
   STATUS[44].EXT.Forced := FALSE;
   STATUS[44].EXT.BIT29 := FALSE;
   STATUS[44].EXT.BIT30 := FALSE;
   STATUS[44].EXT.BIT31 := FALSE;
   STATUS[44].EXT.ModeBit1 := FALSE;
   STATUS[44].EXT.ModeBit2 := FALSE;
   STATUS[44].EXT.ModeBit3 := FALSE;
   STATUS[44].EXT.BIT19 := FALSE;
   STATUS[44].EXT.BIT20 := FALSE;
   STATUS[44].EXT.AlarmSuppressed := FALSE;
   STATUS[44].EXT.AlarmPresent := FALSE;
   STATUS[44].EXT.AlarmFailUnAck := FALSE;
   STATUS[44].Status := 0;
   STATUS[44].TimeStamp := 16#0000;
   STATUS[45].EXT.AlarmWarnUnAck := FALSE;
   STATUS[45].EXT.AckRequired := FALSE;
   STATUS[45].EXT.Maintanence := FALSE;
   STATUS[45].EXT.Operation := FALSE;
   STATUS[45].EXT.Forced := FALSE;
   STATUS[45].EXT.BIT29 := FALSE;
   STATUS[45].EXT.BIT30 := FALSE;
   STATUS[45].EXT.BIT31 := FALSE;
   STATUS[45].EXT.ModeBit1 := FALSE;
   STATUS[45].EXT.ModeBit2 := FALSE;
   STATUS[45].EXT.ModeBit3 := FALSE;
   STATUS[45].EXT.BIT19 := FALSE;
   STATUS[45].EXT.BIT20 := FALSE;
   STATUS[45].EXT.AlarmSuppressed := FALSE;
   STATUS[45].EXT.AlarmPresent := FALSE;
   STATUS[45].EXT.AlarmFailUnAck := FALSE;
   STATUS[45].Status := 0;
   STATUS[45].TimeStamp := 16#0000;
   STATUS[46].EXT.AlarmWarnUnAck := FALSE;
   STATUS[46].EXT.AckRequired := FALSE;
   STATUS[46].EXT.Maintanence := FALSE;
   STATUS[46].EXT.Operation := FALSE;
   STATUS[46].EXT.Forced := FALSE;
   STATUS[46].EXT.BIT29 := FALSE;
   STATUS[46].EXT.BIT30 := FALSE;
   STATUS[46].EXT.BIT31 := FALSE;
   STATUS[46].EXT.ModeBit1 := FALSE;
   STATUS[46].EXT.ModeBit2 := FALSE;
   STATUS[46].EXT.ModeBit3 := FALSE;
   STATUS[46].EXT.BIT19 := FALSE;
   STATUS[46].EXT.BIT20 := FALSE;
   STATUS[46].EXT.AlarmSuppressed := FALSE;
   STATUS[46].EXT.AlarmPresent := FALSE;
   STATUS[46].EXT.AlarmFailUnAck := FALSE;
   STATUS[46].Status := 0;
   STATUS[46].TimeStamp := 16#0000;
   STATUS[47].EXT.AlarmWarnUnAck := FALSE;
   STATUS[47].EXT.AckRequired := FALSE;
   STATUS[47].EXT.Maintanence := FALSE;
   STATUS[47].EXT.Operation := FALSE;
   STATUS[47].EXT.Forced := FALSE;
   STATUS[47].EXT.BIT29 := FALSE;
   STATUS[47].EXT.BIT30 := FALSE;
   STATUS[47].EXT.BIT31 := FALSE;
   STATUS[47].EXT.ModeBit1 := FALSE;
   STATUS[47].EXT.ModeBit2 := FALSE;
   STATUS[47].EXT.ModeBit3 := FALSE;
   STATUS[47].EXT.BIT19 := FALSE;
   STATUS[47].EXT.BIT20 := FALSE;
   STATUS[47].EXT.AlarmSuppressed := FALSE;
   STATUS[47].EXT.AlarmPresent := FALSE;
   STATUS[47].EXT.AlarmFailUnAck := FALSE;
   STATUS[47].Status := 0;
   STATUS[47].TimeStamp := 16#0000;
   STATUS[48].EXT.AlarmWarnUnAck := FALSE;
   STATUS[48].EXT.AckRequired := FALSE;
   STATUS[48].EXT.Maintanence := FALSE;
   STATUS[48].EXT.Operation := FALSE;
   STATUS[48].EXT.Forced := FALSE;
   STATUS[48].EXT.BIT29 := FALSE;
   STATUS[48].EXT.BIT30 := FALSE;
   STATUS[48].EXT.BIT31 := FALSE;
   STATUS[48].EXT.ModeBit1 := FALSE;
   STATUS[48].EXT.ModeBit2 := FALSE;
   STATUS[48].EXT.ModeBit3 := FALSE;
   STATUS[48].EXT.BIT19 := FALSE;
   STATUS[48].EXT.BIT20 := FALSE;
   STATUS[48].EXT.AlarmSuppressed := FALSE;
   STATUS[48].EXT.AlarmPresent := FALSE;
   STATUS[48].EXT.AlarmFailUnAck := FALSE;
   STATUS[48].Status := 0;
   STATUS[48].TimeStamp := 16#0000;
   STATUS[49].EXT.AlarmWarnUnAck := FALSE;
   STATUS[49].EXT.AckRequired := FALSE;
   STATUS[49].EXT.Maintanence := FALSE;
   STATUS[49].EXT.Operation := FALSE;
   STATUS[49].EXT.Forced := FALSE;
   STATUS[49].EXT.BIT29 := FALSE;
   STATUS[49].EXT.BIT30 := FALSE;
   STATUS[49].EXT.BIT31 := FALSE;
   STATUS[49].EXT.ModeBit1 := FALSE;
   STATUS[49].EXT.ModeBit2 := FALSE;
   STATUS[49].EXT.ModeBit3 := FALSE;
   STATUS[49].EXT.BIT19 := FALSE;
   STATUS[49].EXT.BIT20 := FALSE;
   STATUS[49].EXT.AlarmSuppressed := FALSE;
   STATUS[49].EXT.AlarmPresent := FALSE;
   STATUS[49].EXT.AlarmFailUnAck := FALSE;
   STATUS[49].Status := 0;
   STATUS[49].TimeStamp := 16#0000;
   STATUS[50].EXT.AlarmWarnUnAck := FALSE;
   STATUS[50].EXT.AckRequired := FALSE;
   STATUS[50].EXT.Maintanence := FALSE;
   STATUS[50].EXT.Operation := FALSE;
   STATUS[50].EXT.Forced := FALSE;
   STATUS[50].EXT.BIT29 := FALSE;
   STATUS[50].EXT.BIT30 := FALSE;
   STATUS[50].EXT.BIT31 := FALSE;
   STATUS[50].EXT.ModeBit1 := FALSE;
   STATUS[50].EXT.ModeBit2 := FALSE;
   STATUS[50].EXT.ModeBit3 := FALSE;
   STATUS[50].EXT.BIT19 := FALSE;
   STATUS[50].EXT.BIT20 := FALSE;
   STATUS[50].EXT.AlarmSuppressed := FALSE;
   STATUS[50].EXT.AlarmPresent := FALSE;
   STATUS[50].EXT.AlarmFailUnAck := FALSE;
   STATUS[50].Status := 8193;
   STATUS[50].TimeStamp := 16#6EA7;
   STATUS[51].EXT.AlarmWarnUnAck := FALSE;
   STATUS[51].EXT.AckRequired := FALSE;
   STATUS[51].EXT.Maintanence := FALSE;
   STATUS[51].EXT.Operation := FALSE;
   STATUS[51].EXT.Forced := FALSE;
   STATUS[51].EXT.BIT29 := FALSE;
   STATUS[51].EXT.BIT30 := FALSE;
   STATUS[51].EXT.BIT31 := FALSE;
   STATUS[51].EXT.ModeBit1 := FALSE;
   STATUS[51].EXT.ModeBit2 := FALSE;
   STATUS[51].EXT.ModeBit3 := FALSE;
   STATUS[51].EXT.BIT19 := FALSE;
   STATUS[51].EXT.BIT20 := FALSE;
   STATUS[51].EXT.AlarmSuppressed := FALSE;
   STATUS[51].EXT.AlarmPresent := FALSE;
   STATUS[51].EXT.AlarmFailUnAck := FALSE;
   STATUS[51].Status := 0;
   STATUS[51].TimeStamp := 16#0000;
   STATUS[52].EXT.AlarmWarnUnAck := FALSE;
   STATUS[52].EXT.AckRequired := FALSE;
   STATUS[52].EXT.Maintanence := FALSE;
   STATUS[52].EXT.Operation := FALSE;
   STATUS[52].EXT.Forced := FALSE;
   STATUS[52].EXT.BIT29 := FALSE;
   STATUS[52].EXT.BIT30 := FALSE;
   STATUS[52].EXT.BIT31 := FALSE;
   STATUS[52].EXT.ModeBit1 := FALSE;
   STATUS[52].EXT.ModeBit2 := FALSE;
   STATUS[52].EXT.ModeBit3 := FALSE;
   STATUS[52].EXT.BIT19 := FALSE;
   STATUS[52].EXT.BIT20 := FALSE;
   STATUS[52].EXT.AlarmSuppressed := FALSE;
   STATUS[52].EXT.AlarmPresent := FALSE;
   STATUS[52].EXT.AlarmFailUnAck := FALSE;
   STATUS[52].Status := 0;
   STATUS[52].TimeStamp := 16#0000;
   STATUS[53].EXT.AlarmWarnUnAck := FALSE;
   STATUS[53].EXT.AckRequired := FALSE;
   STATUS[53].EXT.Maintanence := FALSE;
   STATUS[53].EXT.Operation := FALSE;
   STATUS[53].EXT.Forced := FALSE;
   STATUS[53].EXT.BIT29 := FALSE;
   STATUS[53].EXT.BIT30 := FALSE;
   STATUS[53].EXT.BIT31 := FALSE;
   STATUS[53].EXT.ModeBit1 := FALSE;
   STATUS[53].EXT.ModeBit2 := FALSE;
   STATUS[53].EXT.ModeBit3 := FALSE;
   STATUS[53].EXT.BIT19 := FALSE;
   STATUS[53].EXT.BIT20 := FALSE;
   STATUS[53].EXT.AlarmSuppressed := FALSE;
   STATUS[53].EXT.AlarmPresent := FALSE;
   STATUS[53].EXT.AlarmFailUnAck := FALSE;
   STATUS[53].Status := 0;
   STATUS[53].TimeStamp := 16#0000;
   STATUS[54].EXT.AlarmWarnUnAck := FALSE;
   STATUS[54].EXT.AckRequired := FALSE;
   STATUS[54].EXT.Maintanence := FALSE;
   STATUS[54].EXT.Operation := FALSE;
   STATUS[54].EXT.Forced := FALSE;
   STATUS[54].EXT.BIT29 := FALSE;
   STATUS[54].EXT.BIT30 := FALSE;
   STATUS[54].EXT.BIT31 := FALSE;
   STATUS[54].EXT.ModeBit1 := FALSE;
   STATUS[54].EXT.ModeBit2 := FALSE;
   STATUS[54].EXT.ModeBit3 := FALSE;
   STATUS[54].EXT.BIT19 := FALSE;
   STATUS[54].EXT.BIT20 := FALSE;
   STATUS[54].EXT.AlarmSuppressed := FALSE;
   STATUS[54].EXT.AlarmPresent := FALSE;
   STATUS[54].EXT.AlarmFailUnAck := FALSE;
   STATUS[54].Status := 0;
   STATUS[54].TimeStamp := 16#0000;
   STATUS[55].EXT.AlarmWarnUnAck := FALSE;
   STATUS[55].EXT.AckRequired := FALSE;
   STATUS[55].EXT.Maintanence := FALSE;
   STATUS[55].EXT.Operation := FALSE;
   STATUS[55].EXT.Forced := FALSE;
   STATUS[55].EXT.BIT29 := FALSE;
   STATUS[55].EXT.BIT30 := FALSE;
   STATUS[55].EXT.BIT31 := FALSE;
   STATUS[55].EXT.ModeBit1 := FALSE;
   STATUS[55].EXT.ModeBit2 := FALSE;
   STATUS[55].EXT.ModeBit3 := FALSE;
   STATUS[55].EXT.BIT19 := FALSE;
   STATUS[55].EXT.BIT20 := FALSE;
   STATUS[55].EXT.AlarmSuppressed := FALSE;
   STATUS[55].EXT.AlarmPresent := FALSE;
   STATUS[55].EXT.AlarmFailUnAck := FALSE;
   STATUS[55].Status := 0;
   STATUS[55].TimeStamp := 16#0000;
   STATUS[56].EXT.AlarmWarnUnAck := FALSE;
   STATUS[56].EXT.AckRequired := FALSE;
   STATUS[56].EXT.Maintanence := FALSE;
   STATUS[56].EXT.Operation := FALSE;
   STATUS[56].EXT.Forced := FALSE;
   STATUS[56].EXT.BIT29 := FALSE;
   STATUS[56].EXT.BIT30 := FALSE;
   STATUS[56].EXT.BIT31 := FALSE;
   STATUS[56].EXT.ModeBit1 := FALSE;
   STATUS[56].EXT.ModeBit2 := FALSE;
   STATUS[56].EXT.ModeBit3 := FALSE;
   STATUS[56].EXT.BIT19 := FALSE;
   STATUS[56].EXT.BIT20 := FALSE;
   STATUS[56].EXT.AlarmSuppressed := FALSE;
   STATUS[56].EXT.AlarmPresent := FALSE;
   STATUS[56].EXT.AlarmFailUnAck := FALSE;
   STATUS[56].Status := 0;
   STATUS[56].TimeStamp := 16#0000;
   STATUS[57].EXT.AlarmWarnUnAck := FALSE;
   STATUS[57].EXT.AckRequired := FALSE;
   STATUS[57].EXT.Maintanence := FALSE;
   STATUS[57].EXT.Operation := FALSE;
   STATUS[57].EXT.Forced := FALSE;
   STATUS[57].EXT.BIT29 := FALSE;
   STATUS[57].EXT.BIT30 := FALSE;
   STATUS[57].EXT.BIT31 := FALSE;
   STATUS[57].EXT.ModeBit1 := FALSE;
   STATUS[57].EXT.ModeBit2 := FALSE;
   STATUS[57].EXT.ModeBit3 := FALSE;
   STATUS[57].EXT.BIT19 := FALSE;
   STATUS[57].EXT.BIT20 := FALSE;
   STATUS[57].EXT.AlarmSuppressed := FALSE;
   STATUS[57].EXT.AlarmPresent := FALSE;
   STATUS[57].EXT.AlarmFailUnAck := FALSE;
   STATUS[57].Status := 0;
   STATUS[57].TimeStamp := 16#0000;
   STATUS[58].EXT.AlarmWarnUnAck := FALSE;
   STATUS[58].EXT.AckRequired := FALSE;
   STATUS[58].EXT.Maintanence := FALSE;
   STATUS[58].EXT.Operation := FALSE;
   STATUS[58].EXT.Forced := FALSE;
   STATUS[58].EXT.BIT29 := FALSE;
   STATUS[58].EXT.BIT30 := FALSE;
   STATUS[58].EXT.BIT31 := FALSE;
   STATUS[58].EXT.ModeBit1 := FALSE;
   STATUS[58].EXT.ModeBit2 := FALSE;
   STATUS[58].EXT.ModeBit3 := FALSE;
   STATUS[58].EXT.BIT19 := FALSE;
   STATUS[58].EXT.BIT20 := FALSE;
   STATUS[58].EXT.AlarmSuppressed := FALSE;
   STATUS[58].EXT.AlarmPresent := FALSE;
   STATUS[58].EXT.AlarmFailUnAck := FALSE;
   STATUS[58].Status := 0;
   STATUS[58].TimeStamp := 16#0000;
   STATUS[59].EXT.AlarmWarnUnAck := FALSE;
   STATUS[59].EXT.AckRequired := FALSE;
   STATUS[59].EXT.Maintanence := FALSE;
   STATUS[59].EXT.Operation := FALSE;
   STATUS[59].EXT.Forced := FALSE;
   STATUS[59].EXT.BIT29 := FALSE;
   STATUS[59].EXT.BIT30 := FALSE;
   STATUS[59].EXT.BIT31 := FALSE;
   STATUS[59].EXT.ModeBit1 := FALSE;
   STATUS[59].EXT.ModeBit2 := FALSE;
   STATUS[59].EXT.ModeBit3 := FALSE;
   STATUS[59].EXT.BIT19 := FALSE;
   STATUS[59].EXT.BIT20 := FALSE;
   STATUS[59].EXT.AlarmSuppressed := FALSE;
   STATUS[59].EXT.AlarmPresent := FALSE;
   STATUS[59].EXT.AlarmFailUnAck := FALSE;
   STATUS[59].Status := 0;
   STATUS[59].TimeStamp := 16#0000;
   STATUS[60].EXT.AlarmWarnUnAck := FALSE;
   STATUS[60].EXT.AckRequired := FALSE;
   STATUS[60].EXT.Maintanence := FALSE;
   STATUS[60].EXT.Operation := FALSE;
   STATUS[60].EXT.Forced := FALSE;
   STATUS[60].EXT.BIT29 := FALSE;
   STATUS[60].EXT.BIT30 := FALSE;
   STATUS[60].EXT.BIT31 := FALSE;
   STATUS[60].EXT.ModeBit1 := FALSE;
   STATUS[60].EXT.ModeBit2 := FALSE;
   STATUS[60].EXT.ModeBit3 := FALSE;
   STATUS[60].EXT.BIT19 := FALSE;
   STATUS[60].EXT.BIT20 := FALSE;
   STATUS[60].EXT.AlarmSuppressed := FALSE;
   STATUS[60].EXT.AlarmPresent := FALSE;
   STATUS[60].EXT.AlarmFailUnAck := FALSE;
   STATUS[60].Status := 0;
   STATUS[60].TimeStamp := 16#0000;
   STATUS[61].EXT.AlarmWarnUnAck := FALSE;
   STATUS[61].EXT.AckRequired := FALSE;
   STATUS[61].EXT.Maintanence := FALSE;
   STATUS[61].EXT.Operation := FALSE;
   STATUS[61].EXT.Forced := FALSE;
   STATUS[61].EXT.BIT29 := FALSE;
   STATUS[61].EXT.BIT30 := FALSE;
   STATUS[61].EXT.BIT31 := FALSE;
   STATUS[61].EXT.ModeBit1 := FALSE;
   STATUS[61].EXT.ModeBit2 := FALSE;
   STATUS[61].EXT.ModeBit3 := FALSE;
   STATUS[61].EXT.BIT19 := FALSE;
   STATUS[61].EXT.BIT20 := FALSE;
   STATUS[61].EXT.AlarmSuppressed := FALSE;
   STATUS[61].EXT.AlarmPresent := FALSE;
   STATUS[61].EXT.AlarmFailUnAck := FALSE;
   STATUS[61].Status := 0;
   STATUS[61].TimeStamp := 16#0000;
   STATUS[62].EXT.AlarmWarnUnAck := FALSE;
   STATUS[62].EXT.AckRequired := FALSE;
   STATUS[62].EXT.Maintanence := FALSE;
   STATUS[62].EXT.Operation := FALSE;
   STATUS[62].EXT.Forced := FALSE;
   STATUS[62].EXT.BIT29 := FALSE;
   STATUS[62].EXT.BIT30 := FALSE;
   STATUS[62].EXT.BIT31 := FALSE;
   STATUS[62].EXT.ModeBit1 := FALSE;
   STATUS[62].EXT.ModeBit2 := FALSE;
   STATUS[62].EXT.ModeBit3 := FALSE;
   STATUS[62].EXT.BIT19 := FALSE;
   STATUS[62].EXT.BIT20 := FALSE;
   STATUS[62].EXT.AlarmSuppressed := FALSE;
   STATUS[62].EXT.AlarmPresent := FALSE;
   STATUS[62].EXT.AlarmFailUnAck := FALSE;
   STATUS[62].Status := 0;
   STATUS[62].TimeStamp := 16#0000;
   STATUS[63].EXT.AlarmWarnUnAck := FALSE;
   STATUS[63].EXT.AckRequired := FALSE;
   STATUS[63].EXT.Maintanence := FALSE;
   STATUS[63].EXT.Operation := FALSE;
   STATUS[63].EXT.Forced := FALSE;
   STATUS[63].EXT.BIT29 := FALSE;
   STATUS[63].EXT.BIT30 := FALSE;
   STATUS[63].EXT.BIT31 := FALSE;
   STATUS[63].EXT.ModeBit1 := FALSE;
   STATUS[63].EXT.ModeBit2 := FALSE;
   STATUS[63].EXT.ModeBit3 := FALSE;
   STATUS[63].EXT.BIT19 := FALSE;
   STATUS[63].EXT.BIT20 := FALSE;
   STATUS[63].EXT.AlarmSuppressed := FALSE;
   STATUS[63].EXT.AlarmPresent := FALSE;
   STATUS[63].EXT.AlarmFailUnAck := FALSE;
   STATUS[63].Status := 0;
   STATUS[63].TimeStamp := 16#0000;
   STATUS[64].EXT.AlarmWarnUnAck := FALSE;
   STATUS[64].EXT.AckRequired := FALSE;
   STATUS[64].EXT.Maintanence := FALSE;
   STATUS[64].EXT.Operation := FALSE;
   STATUS[64].EXT.Forced := FALSE;
   STATUS[64].EXT.BIT29 := FALSE;
   STATUS[64].EXT.BIT30 := FALSE;
   STATUS[64].EXT.BIT31 := FALSE;
   STATUS[64].EXT.ModeBit1 := FALSE;
   STATUS[64].EXT.ModeBit2 := FALSE;
   STATUS[64].EXT.ModeBit3 := FALSE;
   STATUS[64].EXT.BIT19 := FALSE;
   STATUS[64].EXT.BIT20 := FALSE;
   STATUS[64].EXT.AlarmSuppressed := FALSE;
   STATUS[64].EXT.AlarmPresent := FALSE;
   STATUS[64].EXT.AlarmFailUnAck := FALSE;
   STATUS[64].Status := 0;
   STATUS[64].TimeStamp := 16#0000;
   STATUS[65].EXT.AlarmWarnUnAck := FALSE;
   STATUS[65].EXT.AckRequired := FALSE;
   STATUS[65].EXT.Maintanence := FALSE;
   STATUS[65].EXT.Operation := FALSE;
   STATUS[65].EXT.Forced := FALSE;
   STATUS[65].EXT.BIT29 := FALSE;
   STATUS[65].EXT.BIT30 := FALSE;
   STATUS[65].EXT.BIT31 := FALSE;
   STATUS[65].EXT.ModeBit1 := FALSE;
   STATUS[65].EXT.ModeBit2 := FALSE;
   STATUS[65].EXT.ModeBit3 := FALSE;
   STATUS[65].EXT.BIT19 := FALSE;
   STATUS[65].EXT.BIT20 := FALSE;
   STATUS[65].EXT.AlarmSuppressed := FALSE;
   STATUS[65].EXT.AlarmPresent := FALSE;
   STATUS[65].EXT.AlarmFailUnAck := FALSE;
   STATUS[65].Status := 0;
   STATUS[65].TimeStamp := 16#0000;
   STATUS[66].EXT.AlarmWarnUnAck := FALSE;
   STATUS[66].EXT.AckRequired := FALSE;
   STATUS[66].EXT.Maintanence := FALSE;
   STATUS[66].EXT.Operation := FALSE;
   STATUS[66].EXT.Forced := FALSE;
   STATUS[66].EXT.BIT29 := FALSE;
   STATUS[66].EXT.BIT30 := FALSE;
   STATUS[66].EXT.BIT31 := FALSE;
   STATUS[66].EXT.ModeBit1 := FALSE;
   STATUS[66].EXT.ModeBit2 := FALSE;
   STATUS[66].EXT.ModeBit3 := FALSE;
   STATUS[66].EXT.BIT19 := FALSE;
   STATUS[66].EXT.BIT20 := FALSE;
   STATUS[66].EXT.AlarmSuppressed := FALSE;
   STATUS[66].EXT.AlarmPresent := FALSE;
   STATUS[66].EXT.AlarmFailUnAck := FALSE;
   STATUS[66].Status := 0;
   STATUS[66].TimeStamp := 16#0000;
   STATUS[67].EXT.AlarmWarnUnAck := FALSE;
   STATUS[67].EXT.AckRequired := FALSE;
   STATUS[67].EXT.Maintanence := FALSE;
   STATUS[67].EXT.Operation := FALSE;
   STATUS[67].EXT.Forced := FALSE;
   STATUS[67].EXT.BIT29 := FALSE;
   STATUS[67].EXT.BIT30 := FALSE;
   STATUS[67].EXT.BIT31 := FALSE;
   STATUS[67].EXT.ModeBit1 := FALSE;
   STATUS[67].EXT.ModeBit2 := FALSE;
   STATUS[67].EXT.ModeBit3 := FALSE;
   STATUS[67].EXT.BIT19 := FALSE;
   STATUS[67].EXT.BIT20 := FALSE;
   STATUS[67].EXT.AlarmSuppressed := FALSE;
   STATUS[67].EXT.AlarmPresent := FALSE;
   STATUS[67].EXT.AlarmFailUnAck := FALSE;
   STATUS[67].Status := 0;
   STATUS[67].TimeStamp := 16#0000;
   STATUS[68].EXT.AlarmWarnUnAck := FALSE;
   STATUS[68].EXT.AckRequired := FALSE;
   STATUS[68].EXT.Maintanence := FALSE;
   STATUS[68].EXT.Operation := FALSE;
   STATUS[68].EXT.Forced := FALSE;
   STATUS[68].EXT.BIT29 := FALSE;
   STATUS[68].EXT.BIT30 := FALSE;
   STATUS[68].EXT.BIT31 := FALSE;
   STATUS[68].EXT.ModeBit1 := FALSE;
   STATUS[68].EXT.ModeBit2 := FALSE;
   STATUS[68].EXT.ModeBit3 := FALSE;
   STATUS[68].EXT.BIT19 := FALSE;
   STATUS[68].EXT.BIT20 := FALSE;
   STATUS[68].EXT.AlarmSuppressed := FALSE;
   STATUS[68].EXT.AlarmPresent := FALSE;
   STATUS[68].EXT.AlarmFailUnAck := FALSE;
   STATUS[68].Status := 0;
   STATUS[68].TimeStamp := 16#0000;
   STATUS[69].EXT.AlarmWarnUnAck := FALSE;
   STATUS[69].EXT.AckRequired := FALSE;
   STATUS[69].EXT.Maintanence := FALSE;
   STATUS[69].EXT.Operation := FALSE;
   STATUS[69].EXT.Forced := FALSE;
   STATUS[69].EXT.BIT29 := FALSE;
   STATUS[69].EXT.BIT30 := FALSE;
   STATUS[69].EXT.BIT31 := FALSE;
   STATUS[69].EXT.ModeBit1 := FALSE;
   STATUS[69].EXT.ModeBit2 := FALSE;
   STATUS[69].EXT.ModeBit3 := FALSE;
   STATUS[69].EXT.BIT19 := FALSE;
   STATUS[69].EXT.BIT20 := FALSE;
   STATUS[69].EXT.AlarmSuppressed := FALSE;
   STATUS[69].EXT.AlarmPresent := FALSE;
   STATUS[69].EXT.AlarmFailUnAck := FALSE;
   STATUS[69].Status := 0;
   STATUS[69].TimeStamp := 16#0000;
   STATUS[70].EXT.AlarmWarnUnAck := FALSE;
   STATUS[70].EXT.AckRequired := FALSE;
   STATUS[70].EXT.Maintanence := FALSE;
   STATUS[70].EXT.Operation := FALSE;
   STATUS[70].EXT.Forced := FALSE;
   STATUS[70].EXT.BIT29 := FALSE;
   STATUS[70].EXT.BIT30 := FALSE;
   STATUS[70].EXT.BIT31 := FALSE;
   STATUS[70].EXT.ModeBit1 := FALSE;
   STATUS[70].EXT.ModeBit2 := FALSE;
   STATUS[70].EXT.ModeBit3 := FALSE;
   STATUS[70].EXT.BIT19 := FALSE;
   STATUS[70].EXT.BIT20 := FALSE;
   STATUS[70].EXT.AlarmSuppressed := FALSE;
   STATUS[70].EXT.AlarmPresent := FALSE;
   STATUS[70].EXT.AlarmFailUnAck := FALSE;
   STATUS[70].Status := 0;
   STATUS[70].TimeStamp := 16#0000;
   STATUS[71].EXT.AlarmWarnUnAck := FALSE;
   STATUS[71].EXT.AckRequired := FALSE;
   STATUS[71].EXT.Maintanence := FALSE;
   STATUS[71].EXT.Operation := FALSE;
   STATUS[71].EXT.Forced := FALSE;
   STATUS[71].EXT.BIT29 := FALSE;
   STATUS[71].EXT.BIT30 := FALSE;
   STATUS[71].EXT.BIT31 := FALSE;
   STATUS[71].EXT.ModeBit1 := FALSE;
   STATUS[71].EXT.ModeBit2 := FALSE;
   STATUS[71].EXT.ModeBit3 := FALSE;
   STATUS[71].EXT.BIT19 := FALSE;
   STATUS[71].EXT.BIT20 := FALSE;
   STATUS[71].EXT.AlarmSuppressed := FALSE;
   STATUS[71].EXT.AlarmPresent := FALSE;
   STATUS[71].EXT.AlarmFailUnAck := FALSE;
   STATUS[71].Status := 0;
   STATUS[71].TimeStamp := 16#0000;
   STATUS[72].EXT.AlarmWarnUnAck := FALSE;
   STATUS[72].EXT.AckRequired := FALSE;
   STATUS[72].EXT.Maintanence := FALSE;
   STATUS[72].EXT.Operation := FALSE;
   STATUS[72].EXT.Forced := FALSE;
   STATUS[72].EXT.BIT29 := FALSE;
   STATUS[72].EXT.BIT30 := FALSE;
   STATUS[72].EXT.BIT31 := FALSE;
   STATUS[72].EXT.ModeBit1 := FALSE;
   STATUS[72].EXT.ModeBit2 := FALSE;
   STATUS[72].EXT.ModeBit3 := FALSE;
   STATUS[72].EXT.BIT19 := FALSE;
   STATUS[72].EXT.BIT20 := FALSE;
   STATUS[72].EXT.AlarmSuppressed := FALSE;
   STATUS[72].EXT.AlarmPresent := FALSE;
   STATUS[72].EXT.AlarmFailUnAck := FALSE;
   STATUS[72].Status := 0;
   STATUS[72].TimeStamp := 16#0000;
   STATUS[73].EXT.AlarmWarnUnAck := FALSE;
   STATUS[73].EXT.AckRequired := FALSE;
   STATUS[73].EXT.Maintanence := FALSE;
   STATUS[73].EXT.Operation := FALSE;
   STATUS[73].EXT.Forced := FALSE;
   STATUS[73].EXT.BIT29 := FALSE;
   STATUS[73].EXT.BIT30 := FALSE;
   STATUS[73].EXT.BIT31 := FALSE;
   STATUS[73].EXT.ModeBit1 := FALSE;
   STATUS[73].EXT.ModeBit2 := FALSE;
   STATUS[73].EXT.ModeBit3 := FALSE;
   STATUS[73].EXT.BIT19 := FALSE;
   STATUS[73].EXT.BIT20 := FALSE;
   STATUS[73].EXT.AlarmSuppressed := FALSE;
   STATUS[73].EXT.AlarmPresent := FALSE;
   STATUS[73].EXT.AlarmFailUnAck := FALSE;
   STATUS[73].Status := 0;
   STATUS[73].TimeStamp := 16#0000;
   STATUS[74].EXT.AlarmWarnUnAck := FALSE;
   STATUS[74].EXT.AckRequired := FALSE;
   STATUS[74].EXT.Maintanence := FALSE;
   STATUS[74].EXT.Operation := FALSE;
   STATUS[74].EXT.Forced := FALSE;
   STATUS[74].EXT.BIT29 := FALSE;
   STATUS[74].EXT.BIT30 := FALSE;
   STATUS[74].EXT.BIT31 := FALSE;
   STATUS[74].EXT.ModeBit1 := FALSE;
   STATUS[74].EXT.ModeBit2 := FALSE;
   STATUS[74].EXT.ModeBit3 := FALSE;
   STATUS[74].EXT.BIT19 := FALSE;
   STATUS[74].EXT.BIT20 := FALSE;
   STATUS[74].EXT.AlarmSuppressed := FALSE;
   STATUS[74].EXT.AlarmPresent := FALSE;
   STATUS[74].EXT.AlarmFailUnAck := FALSE;
   STATUS[74].Status := 0;
   STATUS[74].TimeStamp := 16#0000;
   STATUS[75].EXT.AlarmWarnUnAck := FALSE;
   STATUS[75].EXT.AckRequired := FALSE;
   STATUS[75].EXT.Maintanence := FALSE;
   STATUS[75].EXT.Operation := FALSE;
   STATUS[75].EXT.Forced := FALSE;
   STATUS[75].EXT.BIT29 := FALSE;
   STATUS[75].EXT.BIT30 := FALSE;
   STATUS[75].EXT.BIT31 := FALSE;
   STATUS[75].EXT.ModeBit1 := FALSE;
   STATUS[75].EXT.ModeBit2 := FALSE;
   STATUS[75].EXT.ModeBit3 := FALSE;
   STATUS[75].EXT.BIT19 := FALSE;
   STATUS[75].EXT.BIT20 := FALSE;
   STATUS[75].EXT.AlarmSuppressed := FALSE;
   STATUS[75].EXT.AlarmPresent := FALSE;
   STATUS[75].EXT.AlarmFailUnAck := FALSE;
   STATUS[75].Status := 0;
   STATUS[75].TimeStamp := 16#0000;
   STATUS[76].EXT.AlarmWarnUnAck := FALSE;
   STATUS[76].EXT.AckRequired := FALSE;
   STATUS[76].EXT.Maintanence := FALSE;
   STATUS[76].EXT.Operation := FALSE;
   STATUS[76].EXT.Forced := FALSE;
   STATUS[76].EXT.BIT29 := FALSE;
   STATUS[76].EXT.BIT30 := FALSE;
   STATUS[76].EXT.BIT31 := FALSE;
   STATUS[76].EXT.ModeBit1 := FALSE;
   STATUS[76].EXT.ModeBit2 := FALSE;
   STATUS[76].EXT.ModeBit3 := FALSE;
   STATUS[76].EXT.BIT19 := FALSE;
   STATUS[76].EXT.BIT20 := FALSE;
   STATUS[76].EXT.AlarmSuppressed := FALSE;
   STATUS[76].EXT.AlarmPresent := FALSE;
   STATUS[76].EXT.AlarmFailUnAck := FALSE;
   STATUS[76].Status := 0;
   STATUS[76].TimeStamp := 16#0000;
   STATUS[77].EXT.AlarmWarnUnAck := FALSE;
   STATUS[77].EXT.AckRequired := FALSE;
   STATUS[77].EXT.Maintanence := FALSE;
   STATUS[77].EXT.Operation := FALSE;
   STATUS[77].EXT.Forced := FALSE;
   STATUS[77].EXT.BIT29 := FALSE;
   STATUS[77].EXT.BIT30 := FALSE;
   STATUS[77].EXT.BIT31 := FALSE;
   STATUS[77].EXT.ModeBit1 := FALSE;
   STATUS[77].EXT.ModeBit2 := FALSE;
   STATUS[77].EXT.ModeBit3 := FALSE;
   STATUS[77].EXT.BIT19 := FALSE;
   STATUS[77].EXT.BIT20 := FALSE;
   STATUS[77].EXT.AlarmSuppressed := FALSE;
   STATUS[77].EXT.AlarmPresent := FALSE;
   STATUS[77].EXT.AlarmFailUnAck := FALSE;
   STATUS[77].Status := 0;
   STATUS[77].TimeStamp := 16#0000;
   STATUS[78].EXT.AlarmWarnUnAck := FALSE;
   STATUS[78].EXT.AckRequired := FALSE;
   STATUS[78].EXT.Maintanence := FALSE;
   STATUS[78].EXT.Operation := FALSE;
   STATUS[78].EXT.Forced := FALSE;
   STATUS[78].EXT.BIT29 := FALSE;
   STATUS[78].EXT.BIT30 := FALSE;
   STATUS[78].EXT.BIT31 := FALSE;
   STATUS[78].EXT.ModeBit1 := FALSE;
   STATUS[78].EXT.ModeBit2 := FALSE;
   STATUS[78].EXT.ModeBit3 := FALSE;
   STATUS[78].EXT.BIT19 := FALSE;
   STATUS[78].EXT.BIT20 := FALSE;
   STATUS[78].EXT.AlarmSuppressed := FALSE;
   STATUS[78].EXT.AlarmPresent := FALSE;
   STATUS[78].EXT.AlarmFailUnAck := FALSE;
   STATUS[78].Status := 0;
   STATUS[78].TimeStamp := 16#0000;
   STATUS[79].EXT.AlarmWarnUnAck := FALSE;
   STATUS[79].EXT.AckRequired := FALSE;
   STATUS[79].EXT.Maintanence := FALSE;
   STATUS[79].EXT.Operation := FALSE;
   STATUS[79].EXT.Forced := FALSE;
   STATUS[79].EXT.BIT29 := FALSE;
   STATUS[79].EXT.BIT30 := FALSE;
   STATUS[79].EXT.BIT31 := FALSE;
   STATUS[79].EXT.ModeBit1 := FALSE;
   STATUS[79].EXT.ModeBit2 := FALSE;
   STATUS[79].EXT.ModeBit3 := FALSE;
   STATUS[79].EXT.BIT19 := FALSE;
   STATUS[79].EXT.BIT20 := FALSE;
   STATUS[79].EXT.AlarmSuppressed := FALSE;
   STATUS[79].EXT.AlarmPresent := FALSE;
   STATUS[79].EXT.AlarmFailUnAck := FALSE;
   STATUS[79].Status := 0;
   STATUS[79].TimeStamp := 16#0000;
   STATUS[80].EXT.AlarmWarnUnAck := FALSE;
   STATUS[80].EXT.AckRequired := FALSE;
   STATUS[80].EXT.Maintanence := FALSE;
   STATUS[80].EXT.Operation := FALSE;
   STATUS[80].EXT.Forced := FALSE;
   STATUS[80].EXT.BIT29 := FALSE;
   STATUS[80].EXT.BIT30 := FALSE;
   STATUS[80].EXT.BIT31 := FALSE;
   STATUS[80].EXT.ModeBit1 := FALSE;
   STATUS[80].EXT.ModeBit2 := FALSE;
   STATUS[80].EXT.ModeBit3 := FALSE;
   STATUS[80].EXT.BIT19 := FALSE;
   STATUS[80].EXT.BIT20 := FALSE;
   STATUS[80].EXT.AlarmSuppressed := FALSE;
   STATUS[80].EXT.AlarmPresent := FALSE;
   STATUS[80].EXT.AlarmFailUnAck := FALSE;
   STATUS[80].Status := 0;
   STATUS[80].TimeStamp := 16#0000;
   STATUS[81].EXT.AlarmWarnUnAck := FALSE;
   STATUS[81].EXT.AckRequired := FALSE;
   STATUS[81].EXT.Maintanence := FALSE;
   STATUS[81].EXT.Operation := FALSE;
   STATUS[81].EXT.Forced := FALSE;
   STATUS[81].EXT.BIT29 := FALSE;
   STATUS[81].EXT.BIT30 := FALSE;
   STATUS[81].EXT.BIT31 := FALSE;
   STATUS[81].EXT.ModeBit1 := FALSE;
   STATUS[81].EXT.ModeBit2 := FALSE;
   STATUS[81].EXT.ModeBit3 := FALSE;
   STATUS[81].EXT.BIT19 := FALSE;
   STATUS[81].EXT.BIT20 := FALSE;
   STATUS[81].EXT.AlarmSuppressed := FALSE;
   STATUS[81].EXT.AlarmPresent := FALSE;
   STATUS[81].EXT.AlarmFailUnAck := FALSE;
   STATUS[81].Status := 0;
   STATUS[81].TimeStamp := 16#0000;
   STATUS[82].EXT.AlarmWarnUnAck := FALSE;
   STATUS[82].EXT.AckRequired := FALSE;
   STATUS[82].EXT.Maintanence := FALSE;
   STATUS[82].EXT.Operation := FALSE;
   STATUS[82].EXT.Forced := FALSE;
   STATUS[82].EXT.BIT29 := FALSE;
   STATUS[82].EXT.BIT30 := FALSE;
   STATUS[82].EXT.BIT31 := FALSE;
   STATUS[82].EXT.ModeBit1 := FALSE;
   STATUS[82].EXT.ModeBit2 := FALSE;
   STATUS[82].EXT.ModeBit3 := FALSE;
   STATUS[82].EXT.BIT19 := FALSE;
   STATUS[82].EXT.BIT20 := FALSE;
   STATUS[82].EXT.AlarmSuppressed := FALSE;
   STATUS[82].EXT.AlarmPresent := FALSE;
   STATUS[82].EXT.AlarmFailUnAck := FALSE;
   STATUS[82].Status := 0;
   STATUS[82].TimeStamp := 16#0000;
   STATUS[83].EXT.AlarmWarnUnAck := FALSE;
   STATUS[83].EXT.AckRequired := FALSE;
   STATUS[83].EXT.Maintanence := FALSE;
   STATUS[83].EXT.Operation := FALSE;
   STATUS[83].EXT.Forced := FALSE;
   STATUS[83].EXT.BIT29 := FALSE;
   STATUS[83].EXT.BIT30 := FALSE;
   STATUS[83].EXT.BIT31 := FALSE;
   STATUS[83].EXT.ModeBit1 := FALSE;
   STATUS[83].EXT.ModeBit2 := FALSE;
   STATUS[83].EXT.ModeBit3 := FALSE;
   STATUS[83].EXT.BIT19 := FALSE;
   STATUS[83].EXT.BIT20 := FALSE;
   STATUS[83].EXT.AlarmSuppressed := FALSE;
   STATUS[83].EXT.AlarmPresent := FALSE;
   STATUS[83].EXT.AlarmFailUnAck := FALSE;
   STATUS[83].Status := 0;
   STATUS[83].TimeStamp := 16#0000;
   STATUS[84].EXT.AlarmWarnUnAck := FALSE;
   STATUS[84].EXT.AckRequired := FALSE;
   STATUS[84].EXT.Maintanence := FALSE;
   STATUS[84].EXT.Operation := FALSE;
   STATUS[84].EXT.Forced := FALSE;
   STATUS[84].EXT.BIT29 := FALSE;
   STATUS[84].EXT.BIT30 := FALSE;
   STATUS[84].EXT.BIT31 := FALSE;
   STATUS[84].EXT.ModeBit1 := FALSE;
   STATUS[84].EXT.ModeBit2 := FALSE;
   STATUS[84].EXT.ModeBit3 := FALSE;
   STATUS[84].EXT.BIT19 := FALSE;
   STATUS[84].EXT.BIT20 := FALSE;
   STATUS[84].EXT.AlarmSuppressed := FALSE;
   STATUS[84].EXT.AlarmPresent := FALSE;
   STATUS[84].EXT.AlarmFailUnAck := FALSE;
   STATUS[84].Status := 0;
   STATUS[84].TimeStamp := 16#0000;
   STATUS[85].EXT.AlarmWarnUnAck := FALSE;
   STATUS[85].EXT.AckRequired := FALSE;
   STATUS[85].EXT.Maintanence := FALSE;
   STATUS[85].EXT.Operation := FALSE;
   STATUS[85].EXT.Forced := FALSE;
   STATUS[85].EXT.BIT29 := FALSE;
   STATUS[85].EXT.BIT30 := FALSE;
   STATUS[85].EXT.BIT31 := FALSE;
   STATUS[85].EXT.ModeBit1 := FALSE;
   STATUS[85].EXT.ModeBit2 := FALSE;
   STATUS[85].EXT.ModeBit3 := FALSE;
   STATUS[85].EXT.BIT19 := FALSE;
   STATUS[85].EXT.BIT20 := FALSE;
   STATUS[85].EXT.AlarmSuppressed := FALSE;
   STATUS[85].EXT.AlarmPresent := FALSE;
   STATUS[85].EXT.AlarmFailUnAck := FALSE;
   STATUS[85].Status := 0;
   STATUS[85].TimeStamp := 16#0000;
   STATUS[86].EXT.AlarmWarnUnAck := FALSE;
   STATUS[86].EXT.AckRequired := FALSE;
   STATUS[86].EXT.Maintanence := FALSE;
   STATUS[86].EXT.Operation := FALSE;
   STATUS[86].EXT.Forced := FALSE;
   STATUS[86].EXT.BIT29 := FALSE;
   STATUS[86].EXT.BIT30 := FALSE;
   STATUS[86].EXT.BIT31 := FALSE;
   STATUS[86].EXT.ModeBit1 := FALSE;
   STATUS[86].EXT.ModeBit2 := FALSE;
   STATUS[86].EXT.ModeBit3 := FALSE;
   STATUS[86].EXT.BIT19 := FALSE;
   STATUS[86].EXT.BIT20 := FALSE;
   STATUS[86].EXT.AlarmSuppressed := FALSE;
   STATUS[86].EXT.AlarmPresent := FALSE;
   STATUS[86].EXT.AlarmFailUnAck := FALSE;
   STATUS[86].Status := 0;
   STATUS[86].TimeStamp := 16#0000;
   STATUS[87].EXT.AlarmWarnUnAck := FALSE;
   STATUS[87].EXT.AckRequired := FALSE;
   STATUS[87].EXT.Maintanence := FALSE;
   STATUS[87].EXT.Operation := FALSE;
   STATUS[87].EXT.Forced := FALSE;
   STATUS[87].EXT.BIT29 := FALSE;
   STATUS[87].EXT.BIT30 := FALSE;
   STATUS[87].EXT.BIT31 := FALSE;
   STATUS[87].EXT.ModeBit1 := FALSE;
   STATUS[87].EXT.ModeBit2 := FALSE;
   STATUS[87].EXT.ModeBit3 := FALSE;
   STATUS[87].EXT.BIT19 := FALSE;
   STATUS[87].EXT.BIT20 := FALSE;
   STATUS[87].EXT.AlarmSuppressed := FALSE;
   STATUS[87].EXT.AlarmPresent := FALSE;
   STATUS[87].EXT.AlarmFailUnAck := FALSE;
   STATUS[87].Status := 0;
   STATUS[87].TimeStamp := 16#0000;
   STATUS[88].EXT.AlarmWarnUnAck := FALSE;
   STATUS[88].EXT.AckRequired := FALSE;
   STATUS[88].EXT.Maintanence := FALSE;
   STATUS[88].EXT.Operation := FALSE;
   STATUS[88].EXT.Forced := FALSE;
   STATUS[88].EXT.BIT29 := FALSE;
   STATUS[88].EXT.BIT30 := FALSE;
   STATUS[88].EXT.BIT31 := FALSE;
   STATUS[88].EXT.ModeBit1 := FALSE;
   STATUS[88].EXT.ModeBit2 := FALSE;
   STATUS[88].EXT.ModeBit3 := FALSE;
   STATUS[88].EXT.BIT19 := FALSE;
   STATUS[88].EXT.BIT20 := FALSE;
   STATUS[88].EXT.AlarmSuppressed := FALSE;
   STATUS[88].EXT.AlarmPresent := FALSE;
   STATUS[88].EXT.AlarmFailUnAck := FALSE;
   STATUS[88].Status := 0;
   STATUS[88].TimeStamp := 16#0000;
   STATUS[89].EXT.AlarmWarnUnAck := FALSE;
   STATUS[89].EXT.AckRequired := FALSE;
   STATUS[89].EXT.Maintanence := FALSE;
   STATUS[89].EXT.Operation := FALSE;
   STATUS[89].EXT.Forced := FALSE;
   STATUS[89].EXT.BIT29 := FALSE;
   STATUS[89].EXT.BIT30 := FALSE;
   STATUS[89].EXT.BIT31 := FALSE;
   STATUS[89].EXT.ModeBit1 := FALSE;
   STATUS[89].EXT.ModeBit2 := FALSE;
   STATUS[89].EXT.ModeBit3 := FALSE;
   STATUS[89].EXT.BIT19 := FALSE;
   STATUS[89].EXT.BIT20 := FALSE;
   STATUS[89].EXT.AlarmSuppressed := FALSE;
   STATUS[89].EXT.AlarmPresent := FALSE;
   STATUS[89].EXT.AlarmFailUnAck := FALSE;
   STATUS[89].Status := 0;
   STATUS[89].TimeStamp := 16#0000;
   STATUS[90].EXT.AlarmWarnUnAck := FALSE;
   STATUS[90].EXT.AckRequired := FALSE;
   STATUS[90].EXT.Maintanence := FALSE;
   STATUS[90].EXT.Operation := FALSE;
   STATUS[90].EXT.Forced := FALSE;
   STATUS[90].EXT.BIT29 := FALSE;
   STATUS[90].EXT.BIT30 := FALSE;
   STATUS[90].EXT.BIT31 := FALSE;
   STATUS[90].EXT.ModeBit1 := FALSE;
   STATUS[90].EXT.ModeBit2 := FALSE;
   STATUS[90].EXT.ModeBit3 := FALSE;
   STATUS[90].EXT.BIT19 := FALSE;
   STATUS[90].EXT.BIT20 := FALSE;
   STATUS[90].EXT.AlarmSuppressed := FALSE;
   STATUS[90].EXT.AlarmPresent := FALSE;
   STATUS[90].EXT.AlarmFailUnAck := FALSE;
   STATUS[90].Status := 0;
   STATUS[90].TimeStamp := 16#0000;
   STATUS[91].EXT.AlarmWarnUnAck := FALSE;
   STATUS[91].EXT.AckRequired := FALSE;
   STATUS[91].EXT.Maintanence := FALSE;
   STATUS[91].EXT.Operation := FALSE;
   STATUS[91].EXT.Forced := FALSE;
   STATUS[91].EXT.BIT29 := FALSE;
   STATUS[91].EXT.BIT30 := FALSE;
   STATUS[91].EXT.BIT31 := FALSE;
   STATUS[91].EXT.ModeBit1 := FALSE;
   STATUS[91].EXT.ModeBit2 := FALSE;
   STATUS[91].EXT.ModeBit3 := FALSE;
   STATUS[91].EXT.BIT19 := FALSE;
   STATUS[91].EXT.BIT20 := FALSE;
   STATUS[91].EXT.AlarmSuppressed := FALSE;
   STATUS[91].EXT.AlarmPresent := FALSE;
   STATUS[91].EXT.AlarmFailUnAck := FALSE;
   STATUS[91].Status := 0;
   STATUS[91].TimeStamp := 16#0000;
   STATUS[92].EXT.AlarmWarnUnAck := FALSE;
   STATUS[92].EXT.AckRequired := FALSE;
   STATUS[92].EXT.Maintanence := FALSE;
   STATUS[92].EXT.Operation := FALSE;
   STATUS[92].EXT.Forced := FALSE;
   STATUS[92].EXT.BIT29 := FALSE;
   STATUS[92].EXT.BIT30 := FALSE;
   STATUS[92].EXT.BIT31 := FALSE;
   STATUS[92].EXT.ModeBit1 := FALSE;
   STATUS[92].EXT.ModeBit2 := FALSE;
   STATUS[92].EXT.ModeBit3 := FALSE;
   STATUS[92].EXT.BIT19 := FALSE;
   STATUS[92].EXT.BIT20 := FALSE;
   STATUS[92].EXT.AlarmSuppressed := FALSE;
   STATUS[92].EXT.AlarmPresent := FALSE;
   STATUS[92].EXT.AlarmFailUnAck := FALSE;
   STATUS[92].Status := 0;
   STATUS[92].TimeStamp := 16#0000;
   STATUS[93].EXT.AlarmWarnUnAck := FALSE;
   STATUS[93].EXT.AckRequired := FALSE;
   STATUS[93].EXT.Maintanence := FALSE;
   STATUS[93].EXT.Operation := FALSE;
   STATUS[93].EXT.Forced := FALSE;
   STATUS[93].EXT.BIT29 := FALSE;
   STATUS[93].EXT.BIT30 := FALSE;
   STATUS[93].EXT.BIT31 := FALSE;
   STATUS[93].EXT.ModeBit1 := FALSE;
   STATUS[93].EXT.ModeBit2 := FALSE;
   STATUS[93].EXT.ModeBit3 := FALSE;
   STATUS[93].EXT.BIT19 := FALSE;
   STATUS[93].EXT.BIT20 := FALSE;
   STATUS[93].EXT.AlarmSuppressed := FALSE;
   STATUS[93].EXT.AlarmPresent := FALSE;
   STATUS[93].EXT.AlarmFailUnAck := FALSE;
   STATUS[93].Status := 0;
   STATUS[93].TimeStamp := 16#0000;
   STATUS[94].EXT.AlarmWarnUnAck := FALSE;
   STATUS[94].EXT.AckRequired := FALSE;
   STATUS[94].EXT.Maintanence := FALSE;
   STATUS[94].EXT.Operation := FALSE;
   STATUS[94].EXT.Forced := FALSE;
   STATUS[94].EXT.BIT29 := FALSE;
   STATUS[94].EXT.BIT30 := FALSE;
   STATUS[94].EXT.BIT31 := FALSE;
   STATUS[94].EXT.ModeBit1 := FALSE;
   STATUS[94].EXT.ModeBit2 := FALSE;
   STATUS[94].EXT.ModeBit3 := FALSE;
   STATUS[94].EXT.BIT19 := FALSE;
   STATUS[94].EXT.BIT20 := FALSE;
   STATUS[94].EXT.AlarmSuppressed := FALSE;
   STATUS[94].EXT.AlarmPresent := FALSE;
   STATUS[94].EXT.AlarmFailUnAck := FALSE;
   STATUS[94].Status := 0;
   STATUS[94].TimeStamp := 16#0000;
   STATUS[95].EXT.AlarmWarnUnAck := FALSE;
   STATUS[95].EXT.AckRequired := FALSE;
   STATUS[95].EXT.Maintanence := FALSE;
   STATUS[95].EXT.Operation := FALSE;
   STATUS[95].EXT.Forced := FALSE;
   STATUS[95].EXT.BIT29 := FALSE;
   STATUS[95].EXT.BIT30 := FALSE;
   STATUS[95].EXT.BIT31 := FALSE;
   STATUS[95].EXT.ModeBit1 := FALSE;
   STATUS[95].EXT.ModeBit2 := FALSE;
   STATUS[95].EXT.ModeBit3 := FALSE;
   STATUS[95].EXT.BIT19 := FALSE;
   STATUS[95].EXT.BIT20 := FALSE;
   STATUS[95].EXT.AlarmSuppressed := FALSE;
   STATUS[95].EXT.AlarmPresent := FALSE;
   STATUS[95].EXT.AlarmFailUnAck := FALSE;
   STATUS[95].Status := 0;
   STATUS[95].TimeStamp := 16#0000;
   STATUS[96].EXT.AlarmWarnUnAck := FALSE;
   STATUS[96].EXT.AckRequired := FALSE;
   STATUS[96].EXT.Maintanence := FALSE;
   STATUS[96].EXT.Operation := FALSE;
   STATUS[96].EXT.Forced := FALSE;
   STATUS[96].EXT.BIT29 := FALSE;
   STATUS[96].EXT.BIT30 := FALSE;
   STATUS[96].EXT.BIT31 := FALSE;
   STATUS[96].EXT.ModeBit1 := FALSE;
   STATUS[96].EXT.ModeBit2 := FALSE;
   STATUS[96].EXT.ModeBit3 := FALSE;
   STATUS[96].EXT.BIT19 := FALSE;
   STATUS[96].EXT.BIT20 := FALSE;
   STATUS[96].EXT.AlarmSuppressed := FALSE;
   STATUS[96].EXT.AlarmPresent := FALSE;
   STATUS[96].EXT.AlarmFailUnAck := FALSE;
   STATUS[96].Status := 0;
   STATUS[96].TimeStamp := 16#0000;
   STATUS[97].EXT.AlarmWarnUnAck := FALSE;
   STATUS[97].EXT.AckRequired := FALSE;
   STATUS[97].EXT.Maintanence := FALSE;
   STATUS[97].EXT.Operation := FALSE;
   STATUS[97].EXT.Forced := FALSE;
   STATUS[97].EXT.BIT29 := FALSE;
   STATUS[97].EXT.BIT30 := FALSE;
   STATUS[97].EXT.BIT31 := FALSE;
   STATUS[97].EXT.ModeBit1 := FALSE;
   STATUS[97].EXT.ModeBit2 := FALSE;
   STATUS[97].EXT.ModeBit3 := FALSE;
   STATUS[97].EXT.BIT19 := FALSE;
   STATUS[97].EXT.BIT20 := FALSE;
   STATUS[97].EXT.AlarmSuppressed := FALSE;
   STATUS[97].EXT.AlarmPresent := FALSE;
   STATUS[97].EXT.AlarmFailUnAck := FALSE;
   STATUS[97].Status := 0;
   STATUS[97].TimeStamp := 16#0000;
   STATUS[98].EXT.AlarmWarnUnAck := FALSE;
   STATUS[98].EXT.AckRequired := FALSE;
   STATUS[98].EXT.Maintanence := FALSE;
   STATUS[98].EXT.Operation := FALSE;
   STATUS[98].EXT.Forced := FALSE;
   STATUS[98].EXT.BIT29 := FALSE;
   STATUS[98].EXT.BIT30 := FALSE;
   STATUS[98].EXT.BIT31 := FALSE;
   STATUS[98].EXT.ModeBit1 := FALSE;
   STATUS[98].EXT.ModeBit2 := FALSE;
   STATUS[98].EXT.ModeBit3 := FALSE;
   STATUS[98].EXT.BIT19 := FALSE;
   STATUS[98].EXT.BIT20 := FALSE;
   STATUS[98].EXT.AlarmSuppressed := FALSE;
   STATUS[98].EXT.AlarmPresent := FALSE;
   STATUS[98].EXT.AlarmFailUnAck := FALSE;
   STATUS[98].Status := 0;
   STATUS[98].TimeStamp := 16#0000;
   STATUS[99].EXT.AlarmWarnUnAck := FALSE;
   STATUS[99].EXT.AckRequired := FALSE;
   STATUS[99].EXT.Maintanence := FALSE;
   STATUS[99].EXT.Operation := FALSE;
   STATUS[99].EXT.Forced := FALSE;
   STATUS[99].EXT.BIT29 := FALSE;
   STATUS[99].EXT.BIT30 := FALSE;
   STATUS[99].EXT.BIT31 := FALSE;
   STATUS[99].EXT.ModeBit1 := FALSE;
   STATUS[99].EXT.ModeBit2 := FALSE;
   STATUS[99].EXT.ModeBit3 := FALSE;
   STATUS[99].EXT.BIT19 := FALSE;
   STATUS[99].EXT.BIT20 := FALSE;
   STATUS[99].EXT.AlarmSuppressed := FALSE;
   STATUS[99].EXT.AlarmPresent := FALSE;
   STATUS[99].EXT.AlarmFailUnAck := FALSE;
   STATUS[99].Status := 0;
   STATUS[99].TimeStamp := 16#0000;
   STATUS[100].EXT.AlarmWarnUnAck := FALSE;
   STATUS[100].EXT.AckRequired := FALSE;
   STATUS[100].EXT.Maintanence := FALSE;
   STATUS[100].EXT.Operation := FALSE;
   STATUS[100].EXT.Forced := FALSE;
   STATUS[100].EXT.BIT29 := FALSE;
   STATUS[100].EXT.BIT30 := FALSE;
   STATUS[100].EXT.BIT31 := FALSE;
   STATUS[100].EXT.ModeBit1 := FALSE;
   STATUS[100].EXT.ModeBit2 := FALSE;
   STATUS[100].EXT.ModeBit3 := FALSE;
   STATUS[100].EXT.BIT19 := FALSE;
   STATUS[100].EXT.BIT20 := FALSE;
   STATUS[100].EXT.AlarmSuppressed := FALSE;
   STATUS[100].EXT.AlarmPresent := FALSE;
   STATUS[100].EXT.AlarmFailUnAck := FALSE;
   STATUS[100].Status := 0;
   STATUS[100].TimeStamp := 16#0000;
   STATUS[101].EXT.AlarmWarnUnAck := FALSE;
   STATUS[101].EXT.AckRequired := FALSE;
   STATUS[101].EXT.Maintanence := FALSE;
   STATUS[101].EXT.Operation := FALSE;
   STATUS[101].EXT.Forced := FALSE;
   STATUS[101].EXT.BIT29 := FALSE;
   STATUS[101].EXT.BIT30 := FALSE;
   STATUS[101].EXT.BIT31 := FALSE;
   STATUS[101].EXT.ModeBit1 := FALSE;
   STATUS[101].EXT.ModeBit2 := FALSE;
   STATUS[101].EXT.ModeBit3 := FALSE;
   STATUS[101].EXT.BIT19 := FALSE;
   STATUS[101].EXT.BIT20 := FALSE;
   STATUS[101].EXT.AlarmSuppressed := FALSE;
   STATUS[101].EXT.AlarmPresent := FALSE;
   STATUS[101].EXT.AlarmFailUnAck := FALSE;
   STATUS[101].Status := 0;
   STATUS[101].TimeStamp := 16#0000;
   STATUS[102].EXT.AlarmWarnUnAck := FALSE;
   STATUS[102].EXT.AckRequired := FALSE;
   STATUS[102].EXT.Maintanence := FALSE;
   STATUS[102].EXT.Operation := FALSE;
   STATUS[102].EXT.Forced := FALSE;
   STATUS[102].EXT.BIT29 := FALSE;
   STATUS[102].EXT.BIT30 := FALSE;
   STATUS[102].EXT.BIT31 := FALSE;
   STATUS[102].EXT.ModeBit1 := FALSE;
   STATUS[102].EXT.ModeBit2 := FALSE;
   STATUS[102].EXT.ModeBit3 := FALSE;
   STATUS[102].EXT.BIT19 := FALSE;
   STATUS[102].EXT.BIT20 := FALSE;
   STATUS[102].EXT.AlarmSuppressed := FALSE;
   STATUS[102].EXT.AlarmPresent := FALSE;
   STATUS[102].EXT.AlarmFailUnAck := FALSE;
   STATUS[102].Status := 0;
   STATUS[102].TimeStamp := 16#0000;
   STATUS[103].EXT.AlarmWarnUnAck := FALSE;
   STATUS[103].EXT.AckRequired := FALSE;
   STATUS[103].EXT.Maintanence := FALSE;
   STATUS[103].EXT.Operation := FALSE;
   STATUS[103].EXT.Forced := FALSE;
   STATUS[103].EXT.BIT29 := FALSE;
   STATUS[103].EXT.BIT30 := FALSE;
   STATUS[103].EXT.BIT31 := FALSE;
   STATUS[103].EXT.ModeBit1 := FALSE;
   STATUS[103].EXT.ModeBit2 := FALSE;
   STATUS[103].EXT.ModeBit3 := FALSE;
   STATUS[103].EXT.BIT19 := FALSE;
   STATUS[103].EXT.BIT20 := FALSE;
   STATUS[103].EXT.AlarmSuppressed := FALSE;
   STATUS[103].EXT.AlarmPresent := FALSE;
   STATUS[103].EXT.AlarmFailUnAck := FALSE;
   STATUS[103].Status := 0;
   STATUS[103].TimeStamp := 16#0000;
   STATUS[104].EXT.AlarmWarnUnAck := FALSE;
   STATUS[104].EXT.AckRequired := FALSE;
   STATUS[104].EXT.Maintanence := FALSE;
   STATUS[104].EXT.Operation := FALSE;
   STATUS[104].EXT.Forced := FALSE;
   STATUS[104].EXT.BIT29 := FALSE;
   STATUS[104].EXT.BIT30 := FALSE;
   STATUS[104].EXT.BIT31 := FALSE;
   STATUS[104].EXT.ModeBit1 := FALSE;
   STATUS[104].EXT.ModeBit2 := FALSE;
   STATUS[104].EXT.ModeBit3 := FALSE;
   STATUS[104].EXT.BIT19 := FALSE;
   STATUS[104].EXT.BIT20 := FALSE;
   STATUS[104].EXT.AlarmSuppressed := FALSE;
   STATUS[104].EXT.AlarmPresent := FALSE;
   STATUS[104].EXT.AlarmFailUnAck := FALSE;
   STATUS[104].Status := 0;
   STATUS[104].TimeStamp := 16#0000;
   STATUS[105].EXT.AlarmWarnUnAck := FALSE;
   STATUS[105].EXT.AckRequired := FALSE;
   STATUS[105].EXT.Maintanence := FALSE;
   STATUS[105].EXT.Operation := FALSE;
   STATUS[105].EXT.Forced := FALSE;
   STATUS[105].EXT.BIT29 := FALSE;
   STATUS[105].EXT.BIT30 := FALSE;
   STATUS[105].EXT.BIT31 := FALSE;
   STATUS[105].EXT.ModeBit1 := FALSE;
   STATUS[105].EXT.ModeBit2 := FALSE;
   STATUS[105].EXT.ModeBit3 := FALSE;
   STATUS[105].EXT.BIT19 := FALSE;
   STATUS[105].EXT.BIT20 := FALSE;
   STATUS[105].EXT.AlarmSuppressed := FALSE;
   STATUS[105].EXT.AlarmPresent := FALSE;
   STATUS[105].EXT.AlarmFailUnAck := FALSE;
   STATUS[105].Status := 0;
   STATUS[105].TimeStamp := 16#0000;
   STATUS[106].EXT.AlarmWarnUnAck := FALSE;
   STATUS[106].EXT.AckRequired := FALSE;
   STATUS[106].EXT.Maintanence := FALSE;
   STATUS[106].EXT.Operation := FALSE;
   STATUS[106].EXT.Forced := FALSE;
   STATUS[106].EXT.BIT29 := FALSE;
   STATUS[106].EXT.BIT30 := FALSE;
   STATUS[106].EXT.BIT31 := FALSE;
   STATUS[106].EXT.ModeBit1 := FALSE;
   STATUS[106].EXT.ModeBit2 := FALSE;
   STATUS[106].EXT.ModeBit3 := FALSE;
   STATUS[106].EXT.BIT19 := FALSE;
   STATUS[106].EXT.BIT20 := FALSE;
   STATUS[106].EXT.AlarmSuppressed := FALSE;
   STATUS[106].EXT.AlarmPresent := FALSE;
   STATUS[106].EXT.AlarmFailUnAck := FALSE;
   STATUS[106].Status := 0;
   STATUS[106].TimeStamp := 16#0000;
   STATUS[107].EXT.AlarmWarnUnAck := FALSE;
   STATUS[107].EXT.AckRequired := FALSE;
   STATUS[107].EXT.Maintanence := FALSE;
   STATUS[107].EXT.Operation := FALSE;
   STATUS[107].EXT.Forced := FALSE;
   STATUS[107].EXT.BIT29 := FALSE;
   STATUS[107].EXT.BIT30 := FALSE;
   STATUS[107].EXT.BIT31 := FALSE;
   STATUS[107].EXT.ModeBit1 := FALSE;
   STATUS[107].EXT.ModeBit2 := FALSE;
   STATUS[107].EXT.ModeBit3 := FALSE;
   STATUS[107].EXT.BIT19 := FALSE;
   STATUS[107].EXT.BIT20 := FALSE;
   STATUS[107].EXT.AlarmSuppressed := FALSE;
   STATUS[107].EXT.AlarmPresent := FALSE;
   STATUS[107].EXT.AlarmFailUnAck := FALSE;
   STATUS[107].Status := 0;
   STATUS[107].TimeStamp := 16#0000;
   STATUS[108].EXT.AlarmWarnUnAck := FALSE;
   STATUS[108].EXT.AckRequired := FALSE;
   STATUS[108].EXT.Maintanence := FALSE;
   STATUS[108].EXT.Operation := FALSE;
   STATUS[108].EXT.Forced := FALSE;
   STATUS[108].EXT.BIT29 := FALSE;
   STATUS[108].EXT.BIT30 := FALSE;
   STATUS[108].EXT.BIT31 := FALSE;
   STATUS[108].EXT.ModeBit1 := FALSE;
   STATUS[108].EXT.ModeBit2 := FALSE;
   STATUS[108].EXT.ModeBit3 := FALSE;
   STATUS[108].EXT.BIT19 := FALSE;
   STATUS[108].EXT.BIT20 := FALSE;
   STATUS[108].EXT.AlarmSuppressed := FALSE;
   STATUS[108].EXT.AlarmPresent := FALSE;
   STATUS[108].EXT.AlarmFailUnAck := FALSE;
   STATUS[108].Status := 0;
   STATUS[108].TimeStamp := 16#0000;
   STATUS[109].EXT.AlarmWarnUnAck := FALSE;
   STATUS[109].EXT.AckRequired := FALSE;
   STATUS[109].EXT.Maintanence := FALSE;
   STATUS[109].EXT.Operation := FALSE;
   STATUS[109].EXT.Forced := FALSE;
   STATUS[109].EXT.BIT29 := FALSE;
   STATUS[109].EXT.BIT30 := FALSE;
   STATUS[109].EXT.BIT31 := FALSE;
   STATUS[109].EXT.ModeBit1 := FALSE;
   STATUS[109].EXT.ModeBit2 := FALSE;
   STATUS[109].EXT.ModeBit3 := FALSE;
   STATUS[109].EXT.BIT19 := FALSE;
   STATUS[109].EXT.BIT20 := FALSE;
   STATUS[109].EXT.AlarmSuppressed := FALSE;
   STATUS[109].EXT.AlarmPresent := FALSE;
   STATUS[109].EXT.AlarmFailUnAck := FALSE;
   STATUS[109].Status := 0;
   STATUS[109].TimeStamp := 16#0000;
   STATUS[110].EXT.AlarmWarnUnAck := FALSE;
   STATUS[110].EXT.AckRequired := FALSE;
   STATUS[110].EXT.Maintanence := FALSE;
   STATUS[110].EXT.Operation := FALSE;
   STATUS[110].EXT.Forced := FALSE;
   STATUS[110].EXT.BIT29 := FALSE;
   STATUS[110].EXT.BIT30 := FALSE;
   STATUS[110].EXT.BIT31 := FALSE;
   STATUS[110].EXT.ModeBit1 := FALSE;
   STATUS[110].EXT.ModeBit2 := FALSE;
   STATUS[110].EXT.ModeBit3 := FALSE;
   STATUS[110].EXT.BIT19 := FALSE;
   STATUS[110].EXT.BIT20 := FALSE;
   STATUS[110].EXT.AlarmSuppressed := FALSE;
   STATUS[110].EXT.AlarmPresent := FALSE;
   STATUS[110].EXT.AlarmFailUnAck := FALSE;
   STATUS[110].Status := 0;
   STATUS[110].TimeStamp := 16#0000;
   STATUS[111].EXT.AlarmWarnUnAck := FALSE;
   STATUS[111].EXT.AckRequired := FALSE;
   STATUS[111].EXT.Maintanence := FALSE;
   STATUS[111].EXT.Operation := FALSE;
   STATUS[111].EXT.Forced := FALSE;
   STATUS[111].EXT.BIT29 := FALSE;
   STATUS[111].EXT.BIT30 := FALSE;
   STATUS[111].EXT.BIT31 := FALSE;
   STATUS[111].EXT.ModeBit1 := FALSE;
   STATUS[111].EXT.ModeBit2 := FALSE;
   STATUS[111].EXT.ModeBit3 := FALSE;
   STATUS[111].EXT.BIT19 := FALSE;
   STATUS[111].EXT.BIT20 := FALSE;
   STATUS[111].EXT.AlarmSuppressed := FALSE;
   STATUS[111].EXT.AlarmPresent := FALSE;
   STATUS[111].EXT.AlarmFailUnAck := FALSE;
   STATUS[111].Status := 0;
   STATUS[111].TimeStamp := 16#0000;
   STATUS[112].EXT.AlarmWarnUnAck := FALSE;
   STATUS[112].EXT.AckRequired := FALSE;
   STATUS[112].EXT.Maintanence := FALSE;
   STATUS[112].EXT.Operation := FALSE;
   STATUS[112].EXT.Forced := FALSE;
   STATUS[112].EXT.BIT29 := FALSE;
   STATUS[112].EXT.BIT30 := FALSE;
   STATUS[112].EXT.BIT31 := FALSE;
   STATUS[112].EXT.ModeBit1 := FALSE;
   STATUS[112].EXT.ModeBit2 := FALSE;
   STATUS[112].EXT.ModeBit3 := FALSE;
   STATUS[112].EXT.BIT19 := FALSE;
   STATUS[112].EXT.BIT20 := FALSE;
   STATUS[112].EXT.AlarmSuppressed := FALSE;
   STATUS[112].EXT.AlarmPresent := FALSE;
   STATUS[112].EXT.AlarmFailUnAck := FALSE;
   STATUS[112].Status := 0;
   STATUS[112].TimeStamp := 16#0000;
   STATUS[113].EXT.AlarmWarnUnAck := FALSE;
   STATUS[113].EXT.AckRequired := FALSE;
   STATUS[113].EXT.Maintanence := FALSE;
   STATUS[113].EXT.Operation := FALSE;
   STATUS[113].EXT.Forced := FALSE;
   STATUS[113].EXT.BIT29 := FALSE;
   STATUS[113].EXT.BIT30 := FALSE;
   STATUS[113].EXT.BIT31 := FALSE;
   STATUS[113].EXT.ModeBit1 := FALSE;
   STATUS[113].EXT.ModeBit2 := FALSE;
   STATUS[113].EXT.ModeBit3 := FALSE;
   STATUS[113].EXT.BIT19 := FALSE;
   STATUS[113].EXT.BIT20 := FALSE;
   STATUS[113].EXT.AlarmSuppressed := FALSE;
   STATUS[113].EXT.AlarmPresent := FALSE;
   STATUS[113].EXT.AlarmFailUnAck := FALSE;
   STATUS[113].Status := 0;
   STATUS[113].TimeStamp := 16#0000;
   STATUS[114].EXT.AlarmWarnUnAck := FALSE;
   STATUS[114].EXT.AckRequired := FALSE;
   STATUS[114].EXT.Maintanence := FALSE;
   STATUS[114].EXT.Operation := FALSE;
   STATUS[114].EXT.Forced := FALSE;
   STATUS[114].EXT.BIT29 := FALSE;
   STATUS[114].EXT.BIT30 := FALSE;
   STATUS[114].EXT.BIT31 := FALSE;
   STATUS[114].EXT.ModeBit1 := FALSE;
   STATUS[114].EXT.ModeBit2 := FALSE;
   STATUS[114].EXT.ModeBit3 := FALSE;
   STATUS[114].EXT.BIT19 := FALSE;
   STATUS[114].EXT.BIT20 := FALSE;
   STATUS[114].EXT.AlarmSuppressed := FALSE;
   STATUS[114].EXT.AlarmPresent := FALSE;
   STATUS[114].EXT.AlarmFailUnAck := FALSE;
   STATUS[114].Status := 0;
   STATUS[114].TimeStamp := 16#0000;
   STATUS[115].EXT.AlarmWarnUnAck := FALSE;
   STATUS[115].EXT.AckRequired := FALSE;
   STATUS[115].EXT.Maintanence := FALSE;
   STATUS[115].EXT.Operation := FALSE;
   STATUS[115].EXT.Forced := FALSE;
   STATUS[115].EXT.BIT29 := FALSE;
   STATUS[115].EXT.BIT30 := FALSE;
   STATUS[115].EXT.BIT31 := FALSE;
   STATUS[115].EXT.ModeBit1 := FALSE;
   STATUS[115].EXT.ModeBit2 := FALSE;
   STATUS[115].EXT.ModeBit3 := FALSE;
   STATUS[115].EXT.BIT19 := FALSE;
   STATUS[115].EXT.BIT20 := FALSE;
   STATUS[115].EXT.AlarmSuppressed := FALSE;
   STATUS[115].EXT.AlarmPresent := FALSE;
   STATUS[115].EXT.AlarmFailUnAck := FALSE;
   STATUS[115].Status := 0;
   STATUS[115].TimeStamp := 16#0000;
   STATUS[116].EXT.AlarmWarnUnAck := FALSE;
   STATUS[116].EXT.AckRequired := FALSE;
   STATUS[116].EXT.Maintanence := FALSE;
   STATUS[116].EXT.Operation := FALSE;
   STATUS[116].EXT.Forced := FALSE;
   STATUS[116].EXT.BIT29 := FALSE;
   STATUS[116].EXT.BIT30 := FALSE;
   STATUS[116].EXT.BIT31 := FALSE;
   STATUS[116].EXT.ModeBit1 := FALSE;
   STATUS[116].EXT.ModeBit2 := FALSE;
   STATUS[116].EXT.ModeBit3 := FALSE;
   STATUS[116].EXT.BIT19 := FALSE;
   STATUS[116].EXT.BIT20 := FALSE;
   STATUS[116].EXT.AlarmSuppressed := FALSE;
   STATUS[116].EXT.AlarmPresent := FALSE;
   STATUS[116].EXT.AlarmFailUnAck := FALSE;
   STATUS[116].Status := 0;
   STATUS[116].TimeStamp := 16#0000;
   STATUS[117].EXT.AlarmWarnUnAck := FALSE;
   STATUS[117].EXT.AckRequired := FALSE;
   STATUS[117].EXT.Maintanence := FALSE;
   STATUS[117].EXT.Operation := FALSE;
   STATUS[117].EXT.Forced := FALSE;
   STATUS[117].EXT.BIT29 := FALSE;
   STATUS[117].EXT.BIT30 := FALSE;
   STATUS[117].EXT.BIT31 := FALSE;
   STATUS[117].EXT.ModeBit1 := FALSE;
   STATUS[117].EXT.ModeBit2 := FALSE;
   STATUS[117].EXT.ModeBit3 := FALSE;
   STATUS[117].EXT.BIT19 := FALSE;
   STATUS[117].EXT.BIT20 := FALSE;
   STATUS[117].EXT.AlarmSuppressed := FALSE;
   STATUS[117].EXT.AlarmPresent := FALSE;
   STATUS[117].EXT.AlarmFailUnAck := FALSE;
   STATUS[117].Status := 0;
   STATUS[117].TimeStamp := 16#0000;
   STATUS[118].EXT.AlarmWarnUnAck := FALSE;
   STATUS[118].EXT.AckRequired := FALSE;
   STATUS[118].EXT.Maintanence := FALSE;
   STATUS[118].EXT.Operation := FALSE;
   STATUS[118].EXT.Forced := FALSE;
   STATUS[118].EXT.BIT29 := FALSE;
   STATUS[118].EXT.BIT30 := FALSE;
   STATUS[118].EXT.BIT31 := FALSE;
   STATUS[118].EXT.ModeBit1 := FALSE;
   STATUS[118].EXT.ModeBit2 := FALSE;
   STATUS[118].EXT.ModeBit3 := FALSE;
   STATUS[118].EXT.BIT19 := FALSE;
   STATUS[118].EXT.BIT20 := FALSE;
   STATUS[118].EXT.AlarmSuppressed := FALSE;
   STATUS[118].EXT.AlarmPresent := FALSE;
   STATUS[118].EXT.AlarmFailUnAck := FALSE;
   STATUS[118].Status := 0;
   STATUS[118].TimeStamp := 16#0000;
   STATUS[119].EXT.AlarmWarnUnAck := FALSE;
   STATUS[119].EXT.AckRequired := FALSE;
   STATUS[119].EXT.Maintanence := FALSE;
   STATUS[119].EXT.Operation := FALSE;
   STATUS[119].EXT.Forced := FALSE;
   STATUS[119].EXT.BIT29 := FALSE;
   STATUS[119].EXT.BIT30 := FALSE;
   STATUS[119].EXT.BIT31 := FALSE;
   STATUS[119].EXT.ModeBit1 := FALSE;
   STATUS[119].EXT.ModeBit2 := FALSE;
   STATUS[119].EXT.ModeBit3 := FALSE;
   STATUS[119].EXT.BIT19 := FALSE;
   STATUS[119].EXT.BIT20 := FALSE;
   STATUS[119].EXT.AlarmSuppressed := FALSE;
   STATUS[119].EXT.AlarmPresent := FALSE;
   STATUS[119].EXT.AlarmFailUnAck := FALSE;
   STATUS[119].Status := 0;
   STATUS[119].TimeStamp := 16#0000;
   STATUS[120].EXT.AlarmWarnUnAck := FALSE;
   STATUS[120].EXT.AckRequired := FALSE;
   STATUS[120].EXT.Maintanence := FALSE;
   STATUS[120].EXT.Operation := FALSE;
   STATUS[120].EXT.Forced := FALSE;
   STATUS[120].EXT.BIT29 := FALSE;
   STATUS[120].EXT.BIT30 := FALSE;
   STATUS[120].EXT.BIT31 := FALSE;
   STATUS[120].EXT.ModeBit1 := FALSE;
   STATUS[120].EXT.ModeBit2 := FALSE;
   STATUS[120].EXT.ModeBit3 := FALSE;
   STATUS[120].EXT.BIT19 := FALSE;
   STATUS[120].EXT.BIT20 := FALSE;
   STATUS[120].EXT.AlarmSuppressed := FALSE;
   STATUS[120].EXT.AlarmPresent := FALSE;
   STATUS[120].EXT.AlarmFailUnAck := FALSE;
   STATUS[120].Status := 0;
   STATUS[120].TimeStamp := 16#0000;
   STATUS[121].EXT.AlarmWarnUnAck := FALSE;
   STATUS[121].EXT.AckRequired := FALSE;
   STATUS[121].EXT.Maintanence := FALSE;
   STATUS[121].EXT.Operation := FALSE;
   STATUS[121].EXT.Forced := FALSE;
   STATUS[121].EXT.BIT29 := FALSE;
   STATUS[121].EXT.BIT30 := FALSE;
   STATUS[121].EXT.BIT31 := FALSE;
   STATUS[121].EXT.ModeBit1 := FALSE;
   STATUS[121].EXT.ModeBit2 := FALSE;
   STATUS[121].EXT.ModeBit3 := FALSE;
   STATUS[121].EXT.BIT19 := FALSE;
   STATUS[121].EXT.BIT20 := FALSE;
   STATUS[121].EXT.AlarmSuppressed := FALSE;
   STATUS[121].EXT.AlarmPresent := FALSE;
   STATUS[121].EXT.AlarmFailUnAck := FALSE;
   STATUS[121].Status := 0;
   STATUS[121].TimeStamp := 16#0000;
   STATUS[122].EXT.AlarmWarnUnAck := FALSE;
   STATUS[122].EXT.AckRequired := FALSE;
   STATUS[122].EXT.Maintanence := FALSE;
   STATUS[122].EXT.Operation := FALSE;
   STATUS[122].EXT.Forced := FALSE;
   STATUS[122].EXT.BIT29 := FALSE;
   STATUS[122].EXT.BIT30 := FALSE;
   STATUS[122].EXT.BIT31 := FALSE;
   STATUS[122].EXT.ModeBit1 := FALSE;
   STATUS[122].EXT.ModeBit2 := FALSE;
   STATUS[122].EXT.ModeBit3 := FALSE;
   STATUS[122].EXT.BIT19 := FALSE;
   STATUS[122].EXT.BIT20 := FALSE;
   STATUS[122].EXT.AlarmSuppressed := FALSE;
   STATUS[122].EXT.AlarmPresent := FALSE;
   STATUS[122].EXT.AlarmFailUnAck := FALSE;
   STATUS[122].Status := 0;
   STATUS[122].TimeStamp := 16#0000;
   STATUS[123].EXT.AlarmWarnUnAck := FALSE;
   STATUS[123].EXT.AckRequired := FALSE;
   STATUS[123].EXT.Maintanence := FALSE;
   STATUS[123].EXT.Operation := FALSE;
   STATUS[123].EXT.Forced := FALSE;
   STATUS[123].EXT.BIT29 := FALSE;
   STATUS[123].EXT.BIT30 := FALSE;
   STATUS[123].EXT.BIT31 := FALSE;
   STATUS[123].EXT.ModeBit1 := FALSE;
   STATUS[123].EXT.ModeBit2 := FALSE;
   STATUS[123].EXT.ModeBit3 := FALSE;
   STATUS[123].EXT.BIT19 := FALSE;
   STATUS[123].EXT.BIT20 := FALSE;
   STATUS[123].EXT.AlarmSuppressed := FALSE;
   STATUS[123].EXT.AlarmPresent := FALSE;
   STATUS[123].EXT.AlarmFailUnAck := FALSE;
   STATUS[123].Status := 0;
   STATUS[123].TimeStamp := 16#0000;
   STATUS[124].EXT.AlarmWarnUnAck := FALSE;
   STATUS[124].EXT.AckRequired := FALSE;
   STATUS[124].EXT.Maintanence := FALSE;
   STATUS[124].EXT.Operation := FALSE;
   STATUS[124].EXT.Forced := FALSE;
   STATUS[124].EXT.BIT29 := FALSE;
   STATUS[124].EXT.BIT30 := FALSE;
   STATUS[124].EXT.BIT31 := FALSE;
   STATUS[124].EXT.ModeBit1 := FALSE;
   STATUS[124].EXT.ModeBit2 := FALSE;
   STATUS[124].EXT.ModeBit3 := FALSE;
   STATUS[124].EXT.BIT19 := FALSE;
   STATUS[124].EXT.BIT20 := FALSE;
   STATUS[124].EXT.AlarmSuppressed := FALSE;
   STATUS[124].EXT.AlarmPresent := FALSE;
   STATUS[124].EXT.AlarmFailUnAck := FALSE;
   STATUS[124].Status := 0;
   STATUS[124].TimeStamp := 16#0000;
   STATUS[125].EXT.AlarmWarnUnAck := FALSE;
   STATUS[125].EXT.AckRequired := FALSE;
   STATUS[125].EXT.Maintanence := FALSE;
   STATUS[125].EXT.Operation := FALSE;
   STATUS[125].EXT.Forced := FALSE;
   STATUS[125].EXT.BIT29 := FALSE;
   STATUS[125].EXT.BIT30 := FALSE;
   STATUS[125].EXT.BIT31 := FALSE;
   STATUS[125].EXT.ModeBit1 := FALSE;
   STATUS[125].EXT.ModeBit2 := FALSE;
   STATUS[125].EXT.ModeBit3 := FALSE;
   STATUS[125].EXT.BIT19 := FALSE;
   STATUS[125].EXT.BIT20 := FALSE;
   STATUS[125].EXT.AlarmSuppressed := FALSE;
   STATUS[125].EXT.AlarmPresent := FALSE;
   STATUS[125].EXT.AlarmFailUnAck := FALSE;
   STATUS[125].Status := 0;
   STATUS[125].TimeStamp := 16#0000;
   STATUS[126].EXT.AlarmWarnUnAck := FALSE;
   STATUS[126].EXT.AckRequired := FALSE;
   STATUS[126].EXT.Maintanence := FALSE;
   STATUS[126].EXT.Operation := FALSE;
   STATUS[126].EXT.Forced := FALSE;
   STATUS[126].EXT.BIT29 := FALSE;
   STATUS[126].EXT.BIT30 := FALSE;
   STATUS[126].EXT.BIT31 := FALSE;
   STATUS[126].EXT.ModeBit1 := FALSE;
   STATUS[126].EXT.ModeBit2 := FALSE;
   STATUS[126].EXT.ModeBit3 := FALSE;
   STATUS[126].EXT.BIT19 := FALSE;
   STATUS[126].EXT.BIT20 := FALSE;
   STATUS[126].EXT.AlarmSuppressed := FALSE;
   STATUS[126].EXT.AlarmPresent := FALSE;
   STATUS[126].EXT.AlarmFailUnAck := FALSE;
   STATUS[126].Status := 0;
   STATUS[126].TimeStamp := 16#0000;
   STATUS[127].EXT.AlarmWarnUnAck := FALSE;
   STATUS[127].EXT.AckRequired := FALSE;
   STATUS[127].EXT.Maintanence := FALSE;
   STATUS[127].EXT.Operation := FALSE;
   STATUS[127].EXT.Forced := FALSE;
   STATUS[127].EXT.BIT29 := FALSE;
   STATUS[127].EXT.BIT30 := FALSE;
   STATUS[127].EXT.BIT31 := FALSE;
   STATUS[127].EXT.ModeBit1 := FALSE;
   STATUS[127].EXT.ModeBit2 := FALSE;
   STATUS[127].EXT.ModeBit3 := FALSE;
   STATUS[127].EXT.BIT19 := FALSE;
   STATUS[127].EXT.BIT20 := FALSE;
   STATUS[127].EXT.AlarmSuppressed := FALSE;
   STATUS[127].EXT.AlarmPresent := FALSE;
   STATUS[127].EXT.AlarmFailUnAck := FALSE;
   STATUS[127].Status := 0;
   STATUS[127].TimeStamp := 16#0000;
   STATUS[128].EXT.AlarmWarnUnAck := FALSE;
   STATUS[128].EXT.AckRequired := FALSE;
   STATUS[128].EXT.Maintanence := FALSE;
   STATUS[128].EXT.Operation := FALSE;
   STATUS[128].EXT.Forced := FALSE;
   STATUS[128].EXT.BIT29 := FALSE;
   STATUS[128].EXT.BIT30 := FALSE;
   STATUS[128].EXT.BIT31 := FALSE;
   STATUS[128].EXT.ModeBit1 := FALSE;
   STATUS[128].EXT.ModeBit2 := FALSE;
   STATUS[128].EXT.ModeBit3 := FALSE;
   STATUS[128].EXT.BIT19 := FALSE;
   STATUS[128].EXT.BIT20 := FALSE;
   STATUS[128].EXT.AlarmSuppressed := FALSE;
   STATUS[128].EXT.AlarmPresent := FALSE;
   STATUS[128].EXT.AlarmFailUnAck := FALSE;
   STATUS[128].Status := 0;
   STATUS[128].TimeStamp := 16#0000;
   STATUS[129].EXT.AlarmWarnUnAck := FALSE;
   STATUS[129].EXT.AckRequired := FALSE;
   STATUS[129].EXT.Maintanence := FALSE;
   STATUS[129].EXT.Operation := FALSE;
   STATUS[129].EXT.Forced := FALSE;
   STATUS[129].EXT.BIT29 := FALSE;
   STATUS[129].EXT.BIT30 := FALSE;
   STATUS[129].EXT.BIT31 := FALSE;
   STATUS[129].EXT.ModeBit1 := FALSE;
   STATUS[129].EXT.ModeBit2 := FALSE;
   STATUS[129].EXT.ModeBit3 := FALSE;
   STATUS[129].EXT.BIT19 := FALSE;
   STATUS[129].EXT.BIT20 := FALSE;
   STATUS[129].EXT.AlarmSuppressed := FALSE;
   STATUS[129].EXT.AlarmPresent := FALSE;
   STATUS[129].EXT.AlarmFailUnAck := FALSE;
   STATUS[129].Status := 0;
   STATUS[129].TimeStamp := 16#0000;
   STATUS[130].EXT.AlarmWarnUnAck := FALSE;
   STATUS[130].EXT.AckRequired := FALSE;
   STATUS[130].EXT.Maintanence := FALSE;
   STATUS[130].EXT.Operation := FALSE;
   STATUS[130].EXT.Forced := FALSE;
   STATUS[130].EXT.BIT29 := FALSE;
   STATUS[130].EXT.BIT30 := FALSE;
   STATUS[130].EXT.BIT31 := FALSE;
   STATUS[130].EXT.ModeBit1 := FALSE;
   STATUS[130].EXT.ModeBit2 := FALSE;
   STATUS[130].EXT.ModeBit3 := FALSE;
   STATUS[130].EXT.BIT19 := FALSE;
   STATUS[130].EXT.BIT20 := FALSE;
   STATUS[130].EXT.AlarmSuppressed := FALSE;
   STATUS[130].EXT.AlarmPresent := FALSE;
   STATUS[130].EXT.AlarmFailUnAck := FALSE;
   STATUS[130].Status := 0;
   STATUS[130].TimeStamp := 16#0000;
   STATUS[131].EXT.AlarmWarnUnAck := FALSE;
   STATUS[131].EXT.AckRequired := FALSE;
   STATUS[131].EXT.Maintanence := FALSE;
   STATUS[131].EXT.Operation := FALSE;
   STATUS[131].EXT.Forced := FALSE;
   STATUS[131].EXT.BIT29 := FALSE;
   STATUS[131].EXT.BIT30 := FALSE;
   STATUS[131].EXT.BIT31 := FALSE;
   STATUS[131].EXT.ModeBit1 := FALSE;
   STATUS[131].EXT.ModeBit2 := FALSE;
   STATUS[131].EXT.ModeBit3 := FALSE;
   STATUS[131].EXT.BIT19 := FALSE;
   STATUS[131].EXT.BIT20 := FALSE;
   STATUS[131].EXT.AlarmSuppressed := FALSE;
   STATUS[131].EXT.AlarmPresent := FALSE;
   STATUS[131].EXT.AlarmFailUnAck := FALSE;
   STATUS[131].Status := 0;
   STATUS[131].TimeStamp := 16#0000;
   STATUS[132].EXT.AlarmWarnUnAck := FALSE;
   STATUS[132].EXT.AckRequired := FALSE;
   STATUS[132].EXT.Maintanence := FALSE;
   STATUS[132].EXT.Operation := FALSE;
   STATUS[132].EXT.Forced := FALSE;
   STATUS[132].EXT.BIT29 := FALSE;
   STATUS[132].EXT.BIT30 := FALSE;
   STATUS[132].EXT.BIT31 := FALSE;
   STATUS[132].EXT.ModeBit1 := FALSE;
   STATUS[132].EXT.ModeBit2 := FALSE;
   STATUS[132].EXT.ModeBit3 := FALSE;
   STATUS[132].EXT.BIT19 := FALSE;
   STATUS[132].EXT.BIT20 := FALSE;
   STATUS[132].EXT.AlarmSuppressed := FALSE;
   STATUS[132].EXT.AlarmPresent := FALSE;
   STATUS[132].EXT.AlarmFailUnAck := FALSE;
   STATUS[132].Status := 0;
   STATUS[132].TimeStamp := 16#0000;
   STATUS[133].EXT.AlarmWarnUnAck := FALSE;
   STATUS[133].EXT.AckRequired := FALSE;
   STATUS[133].EXT.Maintanence := FALSE;
   STATUS[133].EXT.Operation := FALSE;
   STATUS[133].EXT.Forced := FALSE;
   STATUS[133].EXT.BIT29 := FALSE;
   STATUS[133].EXT.BIT30 := FALSE;
   STATUS[133].EXT.BIT31 := FALSE;
   STATUS[133].EXT.ModeBit1 := FALSE;
   STATUS[133].EXT.ModeBit2 := FALSE;
   STATUS[133].EXT.ModeBit3 := FALSE;
   STATUS[133].EXT.BIT19 := FALSE;
   STATUS[133].EXT.BIT20 := FALSE;
   STATUS[133].EXT.AlarmSuppressed := FALSE;
   STATUS[133].EXT.AlarmPresent := FALSE;
   STATUS[133].EXT.AlarmFailUnAck := FALSE;
   STATUS[133].Status := 0;
   STATUS[133].TimeStamp := 16#0000;
   STATUS[134].EXT.AlarmWarnUnAck := FALSE;
   STATUS[134].EXT.AckRequired := FALSE;
   STATUS[134].EXT.Maintanence := FALSE;
   STATUS[134].EXT.Operation := FALSE;
   STATUS[134].EXT.Forced := FALSE;
   STATUS[134].EXT.BIT29 := FALSE;
   STATUS[134].EXT.BIT30 := FALSE;
   STATUS[134].EXT.BIT31 := FALSE;
   STATUS[134].EXT.ModeBit1 := FALSE;
   STATUS[134].EXT.ModeBit2 := FALSE;
   STATUS[134].EXT.ModeBit3 := FALSE;
   STATUS[134].EXT.BIT19 := FALSE;
   STATUS[134].EXT.BIT20 := FALSE;
   STATUS[134].EXT.AlarmSuppressed := FALSE;
   STATUS[134].EXT.AlarmPresent := FALSE;
   STATUS[134].EXT.AlarmFailUnAck := FALSE;
   STATUS[134].Status := 0;
   STATUS[134].TimeStamp := 16#0000;
   STATUS[135].EXT.AlarmWarnUnAck := FALSE;
   STATUS[135].EXT.AckRequired := FALSE;
   STATUS[135].EXT.Maintanence := FALSE;
   STATUS[135].EXT.Operation := FALSE;
   STATUS[135].EXT.Forced := FALSE;
   STATUS[135].EXT.BIT29 := FALSE;
   STATUS[135].EXT.BIT30 := FALSE;
   STATUS[135].EXT.BIT31 := FALSE;
   STATUS[135].EXT.ModeBit1 := FALSE;
   STATUS[135].EXT.ModeBit2 := FALSE;
   STATUS[135].EXT.ModeBit3 := FALSE;
   STATUS[135].EXT.BIT19 := FALSE;
   STATUS[135].EXT.BIT20 := FALSE;
   STATUS[135].EXT.AlarmSuppressed := FALSE;
   STATUS[135].EXT.AlarmPresent := FALSE;
   STATUS[135].EXT.AlarmFailUnAck := FALSE;
   STATUS[135].Status := 0;
   STATUS[135].TimeStamp := 16#0000;
   STATUS[136].EXT.AlarmWarnUnAck := FALSE;
   STATUS[136].EXT.AckRequired := FALSE;
   STATUS[136].EXT.Maintanence := FALSE;
   STATUS[136].EXT.Operation := FALSE;
   STATUS[136].EXT.Forced := FALSE;
   STATUS[136].EXT.BIT29 := FALSE;
   STATUS[136].EXT.BIT30 := FALSE;
   STATUS[136].EXT.BIT31 := FALSE;
   STATUS[136].EXT.ModeBit1 := FALSE;
   STATUS[136].EXT.ModeBit2 := FALSE;
   STATUS[136].EXT.ModeBit3 := FALSE;
   STATUS[136].EXT.BIT19 := FALSE;
   STATUS[136].EXT.BIT20 := FALSE;
   STATUS[136].EXT.AlarmSuppressed := FALSE;
   STATUS[136].EXT.AlarmPresent := FALSE;
   STATUS[136].EXT.AlarmFailUnAck := FALSE;
   STATUS[136].Status := 0;
   STATUS[136].TimeStamp := 16#0000;
   STATUS[137].EXT.AlarmWarnUnAck := FALSE;
   STATUS[137].EXT.AckRequired := FALSE;
   STATUS[137].EXT.Maintanence := FALSE;
   STATUS[137].EXT.Operation := FALSE;
   STATUS[137].EXT.Forced := FALSE;
   STATUS[137].EXT.BIT29 := FALSE;
   STATUS[137].EXT.BIT30 := FALSE;
   STATUS[137].EXT.BIT31 := FALSE;
   STATUS[137].EXT.ModeBit1 := FALSE;
   STATUS[137].EXT.ModeBit2 := FALSE;
   STATUS[137].EXT.ModeBit3 := FALSE;
   STATUS[137].EXT.BIT19 := FALSE;
   STATUS[137].EXT.BIT20 := FALSE;
   STATUS[137].EXT.AlarmSuppressed := FALSE;
   STATUS[137].EXT.AlarmPresent := FALSE;
   STATUS[137].EXT.AlarmFailUnAck := FALSE;
   STATUS[137].Status := 0;
   STATUS[137].TimeStamp := 16#0000;
   STATUS[138].EXT.AlarmWarnUnAck := FALSE;
   STATUS[138].EXT.AckRequired := FALSE;
   STATUS[138].EXT.Maintanence := FALSE;
   STATUS[138].EXT.Operation := FALSE;
   STATUS[138].EXT.Forced := FALSE;
   STATUS[138].EXT.BIT29 := FALSE;
   STATUS[138].EXT.BIT30 := FALSE;
   STATUS[138].EXT.BIT31 := FALSE;
   STATUS[138].EXT.ModeBit1 := FALSE;
   STATUS[138].EXT.ModeBit2 := FALSE;
   STATUS[138].EXT.ModeBit3 := FALSE;
   STATUS[138].EXT.BIT19 := FALSE;
   STATUS[138].EXT.BIT20 := FALSE;
   STATUS[138].EXT.AlarmSuppressed := FALSE;
   STATUS[138].EXT.AlarmPresent := FALSE;
   STATUS[138].EXT.AlarmFailUnAck := FALSE;
   STATUS[138].Status := 0;
   STATUS[138].TimeStamp := 16#0000;
   STATUS[139].EXT.AlarmWarnUnAck := FALSE;
   STATUS[139].EXT.AckRequired := FALSE;
   STATUS[139].EXT.Maintanence := FALSE;
   STATUS[139].EXT.Operation := FALSE;
   STATUS[139].EXT.Forced := FALSE;
   STATUS[139].EXT.BIT29 := FALSE;
   STATUS[139].EXT.BIT30 := FALSE;
   STATUS[139].EXT.BIT31 := FALSE;
   STATUS[139].EXT.ModeBit1 := FALSE;
   STATUS[139].EXT.ModeBit2 := FALSE;
   STATUS[139].EXT.ModeBit3 := FALSE;
   STATUS[139].EXT.BIT19 := FALSE;
   STATUS[139].EXT.BIT20 := FALSE;
   STATUS[139].EXT.AlarmSuppressed := FALSE;
   STATUS[139].EXT.AlarmPresent := FALSE;
   STATUS[139].EXT.AlarmFailUnAck := FALSE;
   STATUS[139].Status := 0;
   STATUS[139].TimeStamp := 16#0000;
   STATUS[140].EXT.AlarmWarnUnAck := FALSE;
   STATUS[140].EXT.AckRequired := FALSE;
   STATUS[140].EXT.Maintanence := FALSE;
   STATUS[140].EXT.Operation := FALSE;
   STATUS[140].EXT.Forced := FALSE;
   STATUS[140].EXT.BIT29 := FALSE;
   STATUS[140].EXT.BIT30 := FALSE;
   STATUS[140].EXT.BIT31 := FALSE;
   STATUS[140].EXT.ModeBit1 := FALSE;
   STATUS[140].EXT.ModeBit2 := FALSE;
   STATUS[140].EXT.ModeBit3 := FALSE;
   STATUS[140].EXT.BIT19 := FALSE;
   STATUS[140].EXT.BIT20 := FALSE;
   STATUS[140].EXT.AlarmSuppressed := FALSE;
   STATUS[140].EXT.AlarmPresent := FALSE;
   STATUS[140].EXT.AlarmFailUnAck := FALSE;
   STATUS[140].Status := 0;
   STATUS[140].TimeStamp := 16#0000;
   STATUS[141].EXT.AlarmWarnUnAck := FALSE;
   STATUS[141].EXT.AckRequired := FALSE;
   STATUS[141].EXT.Maintanence := FALSE;
   STATUS[141].EXT.Operation := FALSE;
   STATUS[141].EXT.Forced := FALSE;
   STATUS[141].EXT.BIT29 := FALSE;
   STATUS[141].EXT.BIT30 := FALSE;
   STATUS[141].EXT.BIT31 := FALSE;
   STATUS[141].EXT.ModeBit1 := FALSE;
   STATUS[141].EXT.ModeBit2 := FALSE;
   STATUS[141].EXT.ModeBit3 := FALSE;
   STATUS[141].EXT.BIT19 := FALSE;
   STATUS[141].EXT.BIT20 := FALSE;
   STATUS[141].EXT.AlarmSuppressed := FALSE;
   STATUS[141].EXT.AlarmPresent := FALSE;
   STATUS[141].EXT.AlarmFailUnAck := FALSE;
   STATUS[141].Status := 0;
   STATUS[141].TimeStamp := 16#0000;
   STATUS[142].EXT.AlarmWarnUnAck := FALSE;
   STATUS[142].EXT.AckRequired := FALSE;
   STATUS[142].EXT.Maintanence := FALSE;
   STATUS[142].EXT.Operation := FALSE;
   STATUS[142].EXT.Forced := FALSE;
   STATUS[142].EXT.BIT29 := FALSE;
   STATUS[142].EXT.BIT30 := FALSE;
   STATUS[142].EXT.BIT31 := FALSE;
   STATUS[142].EXT.ModeBit1 := FALSE;
   STATUS[142].EXT.ModeBit2 := FALSE;
   STATUS[142].EXT.ModeBit3 := FALSE;
   STATUS[142].EXT.BIT19 := FALSE;
   STATUS[142].EXT.BIT20 := FALSE;
   STATUS[142].EXT.AlarmSuppressed := FALSE;
   STATUS[142].EXT.AlarmPresent := FALSE;
   STATUS[142].EXT.AlarmFailUnAck := FALSE;
   STATUS[142].Status := 0;
   STATUS[142].TimeStamp := 16#0000;
   STATUS[143].EXT.AlarmWarnUnAck := FALSE;
   STATUS[143].EXT.AckRequired := FALSE;
   STATUS[143].EXT.Maintanence := FALSE;
   STATUS[143].EXT.Operation := FALSE;
   STATUS[143].EXT.Forced := FALSE;
   STATUS[143].EXT.BIT29 := FALSE;
   STATUS[143].EXT.BIT30 := FALSE;
   STATUS[143].EXT.BIT31 := FALSE;
   STATUS[143].EXT.ModeBit1 := FALSE;
   STATUS[143].EXT.ModeBit2 := FALSE;
   STATUS[143].EXT.ModeBit3 := FALSE;
   STATUS[143].EXT.BIT19 := FALSE;
   STATUS[143].EXT.BIT20 := FALSE;
   STATUS[143].EXT.AlarmSuppressed := FALSE;
   STATUS[143].EXT.AlarmPresent := FALSE;
   STATUS[143].EXT.AlarmFailUnAck := FALSE;
   STATUS[143].Status := 0;
   STATUS[143].TimeStamp := 16#0000;
   STATUS[144].EXT.AlarmWarnUnAck := FALSE;
   STATUS[144].EXT.AckRequired := FALSE;
   STATUS[144].EXT.Maintanence := FALSE;
   STATUS[144].EXT.Operation := FALSE;
   STATUS[144].EXT.Forced := FALSE;
   STATUS[144].EXT.BIT29 := FALSE;
   STATUS[144].EXT.BIT30 := FALSE;
   STATUS[144].EXT.BIT31 := FALSE;
   STATUS[144].EXT.ModeBit1 := FALSE;
   STATUS[144].EXT.ModeBit2 := FALSE;
   STATUS[144].EXT.ModeBit3 := FALSE;
   STATUS[144].EXT.BIT19 := FALSE;
   STATUS[144].EXT.BIT20 := FALSE;
   STATUS[144].EXT.AlarmSuppressed := FALSE;
   STATUS[144].EXT.AlarmPresent := FALSE;
   STATUS[144].EXT.AlarmFailUnAck := FALSE;
   STATUS[144].Status := 0;
   STATUS[144].TimeStamp := 16#0000;
   STATUS[145].EXT.AlarmWarnUnAck := FALSE;
   STATUS[145].EXT.AckRequired := FALSE;
   STATUS[145].EXT.Maintanence := FALSE;
   STATUS[145].EXT.Operation := FALSE;
   STATUS[145].EXT.Forced := FALSE;
   STATUS[145].EXT.BIT29 := FALSE;
   STATUS[145].EXT.BIT30 := FALSE;
   STATUS[145].EXT.BIT31 := FALSE;
   STATUS[145].EXT.ModeBit1 := FALSE;
   STATUS[145].EXT.ModeBit2 := FALSE;
   STATUS[145].EXT.ModeBit3 := FALSE;
   STATUS[145].EXT.BIT19 := FALSE;
   STATUS[145].EXT.BIT20 := FALSE;
   STATUS[145].EXT.AlarmSuppressed := FALSE;
   STATUS[145].EXT.AlarmPresent := FALSE;
   STATUS[145].EXT.AlarmFailUnAck := FALSE;
   STATUS[145].Status := 0;
   STATUS[145].TimeStamp := 16#0000;
   STATUS[146].EXT.AlarmWarnUnAck := FALSE;
   STATUS[146].EXT.AckRequired := FALSE;
   STATUS[146].EXT.Maintanence := FALSE;
   STATUS[146].EXT.Operation := FALSE;
   STATUS[146].EXT.Forced := FALSE;
   STATUS[146].EXT.BIT29 := FALSE;
   STATUS[146].EXT.BIT30 := FALSE;
   STATUS[146].EXT.BIT31 := FALSE;
   STATUS[146].EXT.ModeBit1 := FALSE;
   STATUS[146].EXT.ModeBit2 := FALSE;
   STATUS[146].EXT.ModeBit3 := FALSE;
   STATUS[146].EXT.BIT19 := FALSE;
   STATUS[146].EXT.BIT20 := FALSE;
   STATUS[146].EXT.AlarmSuppressed := FALSE;
   STATUS[146].EXT.AlarmPresent := FALSE;
   STATUS[146].EXT.AlarmFailUnAck := FALSE;
   STATUS[146].Status := 0;
   STATUS[146].TimeStamp := 16#0000;
   STATUS[147].EXT.AlarmWarnUnAck := FALSE;
   STATUS[147].EXT.AckRequired := FALSE;
   STATUS[147].EXT.Maintanence := FALSE;
   STATUS[147].EXT.Operation := FALSE;
   STATUS[147].EXT.Forced := FALSE;
   STATUS[147].EXT.BIT29 := FALSE;
   STATUS[147].EXT.BIT30 := FALSE;
   STATUS[147].EXT.BIT31 := FALSE;
   STATUS[147].EXT.ModeBit1 := FALSE;
   STATUS[147].EXT.ModeBit2 := FALSE;
   STATUS[147].EXT.ModeBit3 := FALSE;
   STATUS[147].EXT.BIT19 := FALSE;
   STATUS[147].EXT.BIT20 := FALSE;
   STATUS[147].EXT.AlarmSuppressed := FALSE;
   STATUS[147].EXT.AlarmPresent := FALSE;
   STATUS[147].EXT.AlarmFailUnAck := FALSE;
   STATUS[147].Status := 0;
   STATUS[147].TimeStamp := 16#0000;
   STATUS[148].EXT.AlarmWarnUnAck := FALSE;
   STATUS[148].EXT.AckRequired := FALSE;
   STATUS[148].EXT.Maintanence := FALSE;
